	active_fem:				analog_actuator_snapshot;
(*$
	 This message is activated when the active feedback sensor, if present, and  
	analog_actuator <a href="#analog_actuator_status_enum"><i>status</i></a>
 are inchoerent, or it is activated dynamically as a timeout of the activation movement.<br/><br/>
	<a href="#message_behaviour_enum"><i>MESSAGE BEHAVIOUR:</i></a> <i>MESSAGE_BEHAVIOUR_EVENT </i><br/><br/>
	<a href="#machine_reaction_enum"><i>MACHINE REACTION:</i></a> <i>MACHINE_REACTION_NORMAL_STOP </i><br/><br/>
	 The fault codes are specified by ERROR_ID:
	<br/>
	<li> <b>ERRORID_1 = 9</b>: Timeout of activation movement when the <a href="#digital_input_object"><i>di_inactive</i></a>. 
 feedback sensor is covered</li>	
	<li> <b>ERRORID_1 = 10</b>: Timeout of activation movement when the <a href="#digital_input_object"><i>di_ready</i></a>. 
 feedback sensor is not covered</li>	
	<li> <b>ERRORID_1 = 13</b>: Actuator is in <a href="#analog_actuator_status_enum"><i>ANALOG_ACTUATOR_STATUS_ACTIVE</i></a>
 status and the <a href="#digital_input_object"><i>di_ready</i></a> feedback sensor is not covered, or 
 actuator is in <a href="#analog_actuator_status_enum"><i>ANALOG_ACTUATOR_STATUS_INACTIVE</i></a>
 status and the <a href="#digital_input_object"><i>di_ready</i></a> feedback sensor is covered. </li>
$*)

	inactive_fem:			analog_actuator_snapshot;
(*$
	 This message is activated when the inactive feedback sensor, if present, and  
	analog_actuator <a href="#analog_actuator_status_enum"><i>status</i></a>
 are inchoerent, or it is activated dynamically as a timeout of the deactivation movement.<br/><br/>
	<a href="#message_behaviour_enum"><i>MESSAGE BEHAVIOUR:</i></a><i> MESSAGE_BEHAVIOUR_EVENT</i><br/><br/>
	<a href="#machine_reaction_enum"><i>MACHINE REACTION:</i></a><i> MACHINE_REACTION_NORMAL_STOP</i><br/><br/>
	 The fault codes are specified by <i>ERROR_ID</i>:
	<br/>
	<ul>
	<li> <b><i>ERRORID_1 = 11</i></b>: Timeout of deactivation movement when the <a href="#digital_input_object"><i>di_ready</i></a>. 
 feedback sensor is covered</li>	
	<li> <b><i>ERRORID_1 = 12</i></b>: Timeout of deactivation movement when the <a href="#digital_input_object"><i>di_inactive</i></a>. 
 feedback sensor is not covered</li>	
	<li> <b><i>ERRORID_1 = 14</i></b>: Actuator is in <a href="#analog_actuator_status_enum"><i>ANALOG_ACTUATOR_STATUS_INACTIVE</i></a>
 status and the <a href="#digital_input_object"><i>di_inactive</i></a> feedback sensor is not covered, or 
 actuator is in <a href="#analog_actuator_status_enum"><i>ANALOG_ACTUATOR_STATUS_ACTIVE</i></a>
 status and the <a href="#digital_input_object"><i>di_inactive</i></a> feedback sensor is covered. </li>
 </ul>
$*)

	CONVERSION_private:				analog_actuator_private;

    active_elapsed_time: 	LREAL := 0.0;(*$M desc := Elapsed time from the "activate command" and execution finished.; $*)
    deactive_elapsed_time:  LREAL := 0.0;(*$M desc := Elapsed time from the "deactivate command" and execution finished.; $*)

   	ao_setpoint_value: 		LREAL := 0.0;(*$M desc := Analog Output Physical Value; $*)
    ai_feedback_value: 		LREAL := 0.0;(*$M desc := Analog Input Physical Value; $*)

	light_test_active:		BOOL := FALSE;						(*$H_RW desc := Light test is active; $*)

	END_STRUCT
END_TYPE

// ---- Data types/AFL extensions/analog_actuator/analog_actuator_command_enum.TcDUT
TYPE
	analog_actuator_command_enum: (
	ANALOG_ACTUATOR_CMD_NONE			:= 0,	(*$ No command assigned $*)
	ANALOG_ACTUATOR_CMD_INIT			:= 2,	(*$ Initialization command $*)
	ANALOG_ACTUATOR_CMD_ACTIVATE		:= 6,	(*$ Activation command $*)
	ANALOG_ACTUATOR_CMD_DEACTIVATE		:= 8	(*$ Deactivation command $*)
	) := ANALOG_ACTUATOR_CMD_INIT;
END_TYPE

// ---- Data types/AFL extensions/analog_actuator/analog_actuator_fault_reaction_enum.TcDUT
TYPE
	analog_actuator_fault_reaction_enum: (
	ANALOG_ACTUATOR_FAULT_REACTION_DEACTIVATING	:= 0,	(*$ When faulted the analog_actuator sets the
																<a href="#digital_output_object"><i>output</i></a>
																consistently with a deactivate command $*)
	ANALOG_ACTUATOR_FAULT_REACTION_HOLD			:= 1,	(*$ When faulted the analog_actuator sets the
																<a href="#digital_output_object"><i>output</i></a>
																consistently with the current command $*)
	ANALOG_ACTUATOR_FAULT_REACTION_IGNORE		:= 2	(*$ No automatic internal reaction, the application handle the fault condition of analog_actuator $*)
) := ANALOG_ACTUATOR_FAULT_REACTION_DEACTIVATING;
END_TYPE

// ---- Data types/AFL extensions/analog_actuator/analog_actuator_snapshot.TcDUT
(*$S desc := Snapshot; $*)
TYPE
	analog_actuator_snapshot:	STRUCT
	message:        message;

	status:			analog_actuator_status_enum;
	(*$
	Value of the analog_actuator <a href="#analog_actuator_status_enum"><i>status</i></a> field
	when the message is set 
	$*)
	command:		analog_actuator_command_enum;
	(*$
	Value of the analog_actuator <a href="#analog_actuator_command_enum"><i>command</i></a> field
	when the message is set 
	$*)
	is_active:		BOOL;
	(*$
		Value of the active <a href="#digital_input_object"><i>digital_input</i></a>
		when the message is set 
	$*)
	is_inactive:	BOOL;
	(*$
		Value of the inactive <a href="#digital_input_object"><i>digital_input</i></a>
		when the message is set 
	$*)
END_STRUCT
END_TYPE

// ---- Data types/AFL extensions/analog_actuator/analog_actuator_status_enum.TcDUT
(*$ analog_actuator status $*)
TYPE
	analog_actuator_status_enum: (
	ANALOG_ACTUATOR_STATUS_INIT				:= 0,	(*$ analog_actuator initialization $*)
	ANALOG_ACTUATOR_STATUS_ACTIVE 			:= 4,	(*$ analog_actuator is active $*)
	ANALOG_ACTUATOR_STATUS_ACTIVATING		:= 5,	(*$ analog_actuator is executing
														an activation command $*)
	ANALOG_ACTUATOR_STATUS_INACTIVE			:= 6,	(*$ analog_actuator is inactive $*)
	ANALOG_ACTUATOR_STATUS_DEACTIVATING		:= 7,	(*$ analog_actuator is executing
														a deactivation command $*)
	ANALOG_ACTUATOR_STATUS_FAULTED			:= 8	(*$ analog_actuator is in fault status $*)
	) := ANALOG_ACTUATOR_STATUS_INIT;
END_TYPE

// ---- Data types/AFL extensions/analog_actuator/analog_actuator_test.TcDUT
(*$T desc := Test structure; $*)
TYPE
analog_actuator_test:	STRUCT
	command:			analog_actuator_test_command_enum := ANALOG_ACTUATOR_TEST_CMD_IDLE;
															(*$H_W desc := Command (the variable
															  is written by HMI)..; $*)
	command_info:		ARRAY[0..ANALOG_ACTUATOR_MAX_TEST_COMMANDS] OF test_command_info;
															(*$ Structure that informs the HMI
																of the availability of every single
																command and its operational state $*)
    physical_value:		REAL := 0.0;						(*$P min := APPL; max := APPL; step := 0.1;
																 unit := APPL; desc := Analog output physical
																 actual forcing value ; $*)
	
END_STRUCT
END_TYPE

// ---- Data types/AFL extensions/analog_actuator/analog_actuator_test_command_enum.TcDUT
TYPE
	analog_actuator_test_command_enum: (
	ANALOG_ACTUATOR_TEST_CMD_IDLE			:= 0,	(*$ No command assigned $*)
	ANALOG_ACTUATOR_TEST_CMD_ACTIVATE		:= 1,	(*$ Activation command $*)
	ANALOG_ACTUATOR_TEST_CMD_DEACTIVATE		:= 2	(*$ Deactivation command $*)
	) := ANALOG_ACTUATOR_TEST_CMD_IDLE;
END_TYPE

// ---- Data types/AFL extensions/analog_actuator/private/analog_actuator_private.TcDUT
TYPE
	analog_actuator_private :	STRUCT
	initialized:		BOOL := FALSE;		(* The object has been initialized by _init function. *)
	cycle_is_active:	BOOL := FALSE;		(* Cycle function is correctly called. *)
	my_address:			POINTER_TO_VOID; 	(* Object address(pointer).
												Used by HMI for establish
												the objects relations *)

END_STRUCT
END_TYPE

// ---- Data types/AFL extensions/jog_manager/jog_manager.TcDUT
(*   Copyright (c) 2007-2008 G.D SpA
*****************************************************************************************

Date:      Time:     | Author:   				|    Time spent: | Tester:   	   |  Time spent
*****************************************************************************************
*)
(*$
	The <i>jog_manager</i> class abstracts a to manage the axis jog movement.<br/>
	The object is constructed with the <a href="#jog_manager_init"><i>jog_manager_init()</i></a> 
	method and <a href="#axis_object"><i>axi</i></a> are optionally <br/>
	added through the method <a href="#jog_manager_add_axis"><i>jog_manager_add_axis()</i></a>.	
$*)
(* Last used errorID_1 := 15 *)
TYPE
	jog_manager:	STRUCT
	class_name:				STRING(MAX_OBJ_NAME_LENGTH) := JOG_MANAGER_CLASS_NAME;

	object_name:			STRING(MAX_OBJ_NAME_LENGTH) := '';

	descriptor:				descriptor;

	status:					jog_manager_status_enum := JOG_MANAGER_STATUS_INIT;
	(*$M
	desc := Internal status of the jog_manager: value among those defined in the <br/>
	enumerative <a href="#jog_manager_status_enum"><i>jog_manager_status_enum</i></a>; 
	$*)
	command:				jog_manager_command_enum := JOG_MANAGER_CMD_NONE;
												(*$ Command that jog_manager
													is going to execute; value among
													those defined in the enumerative
													jog_manager_command_enum $*)
	operational_command:	jog_manager_command_enum := JOG_MANAGER_CMD_NONE;
												(*$ Command assigned when jog_manager
													is in the "operational" mode; value among
													those defined in the enumerative
													jog_manager_command_enum $*)
	test:					jog_manager_test;
												(*$ This struct contains all the test's informations $*)
	parents:				ARRAY[1..JOG_MANAGER_MAX_PARENTS] OF POINTER TO jog_manager;												
	parents_next_free:		UINT;
												(*$ This array contains all the parent jog_manager $*)
	axis_list:				ARRAY[JOG_MANAGER_JOG_LIST_NONE..JOG_MANAGER_JOG_LIST_MAX] OF jog_manager_element;
												(*$ This struct contains all the axis_jog information $*)
	jog_activation_condition: BOOL;
												(*$ Jog activation condition $*)			
	jog_active:				BOOL;				
	(*$P desc := jog mode active; $*)
	jog_active_pow:			parameter_overwrite;
	(*$I desc := Parameter overwite to inizialithe the value at startup; $*)
	enable_sw_limit:		BOOL;				
	(*$P desc := software limit active; $*)	
	enable_sw_limit_pow:	parameter_overwrite;
	(*$I desc := Parameter overwite to adjust the SW limit check; $*)																										
	axis_act_position_linear: LREAL;
	(*$M unit := mm;
		desc := currently selected axis position; 
	$*)
	axis_act_position_rotative: LREAL;
	(*$M unit := °;
		desc := currently selected axis position; 
	$*)		
	axis_act_torque_rotative: LREAL;
	(*$M unit := %;
		desc := currently selected axis torque (the value is axis indipendent! it's doubled for management reason!; 
	$*)
	axis_act_torque_linear: LREAL;
	(*$M unit := %;
		desc := currently selected axis torque (the value is axis indipendent! it's doubled for management reason!; 
	$*)	
	axis_cmd_position_linear: LREAL;
	(*$P min :=  -1000; max :=  2000; step := 1; unit := mm/s;
		desc := jog command position (linear jog axis); 
	$*)
	axis_cmd_position_rotative:	LREAL;
	(*$P min :=  -360; max :=  360; step := 1; unit := °/s;
		desc := jog command position (rotative jog axis); 
	$*)
	axis_cmd_position_rotative_pow:	parameter_overwrite;
	(*$I desc := Parameter overwite to adjust jog command position (rotative); $*)	
	axis_speed_linear:		LREAL;
	(*$P min :=  0; max :=  100; step := 1; unit := mm/s;
		desc := jog speed (linear jog axis); 
	$*)
	axis_cmd_position_linear_pow: parameter_overwrite;
	(*$I desc := Parameter overwite to adjust jog command position (linear); $*)		
	axis_speed_rotative:	LREAL;
	(*$P min :=  0; max :=  100; step := 1; unit := °/s;
		desc := jog speed (rotative jog axis); 
	$*)	
	di_pendant_positive:	POINTER TO digital_input;
	(*$U
	desc := Reference to the <a href="#digital_input_object"><i>digital_input</i></a>
	which refere to jog positive pendant command; 
	$*)
	di_pendant_negative:	POINTER TO digital_input;
	(*$U
	desc := Reference to the <a href="#digital_input_object"><i>digital_input</i></a>
	which refere to jog negative pendant command; 
	$*)
	has_pendant:			BOOL;
												(*$ Pendant present $*)
	pendant_active:			BOOL;				
	(*$P desc := pendant active; $*)
	pendant_active_pow:		parameter_overwrite;
	(*$I desc := Parameter overwite to inizialithe the value at startup; $*)
	has_shared_pendant:		POINTER TO jog_manager;
	(*$ Pointer to jog_manager instance that manage directly the pendant $*)
	shared_pendant_active:	BOOL;	
	(*$ Shared pendant activation status $*)
								
	hmi_jog_positive_cbtn:	command_button;		(*$I expose{ value_from_hmi; button_status.status; button_led.color; button_led.graphic_object.status;} desc := jog plus; $*)
	hmi_jog_negative_cbtn:	command_button;		(*$I expose{ value_from_hmi; button_status.status; button_led.color; button_led.graphic_object.status;} desc := jog minus; $*)
	hmi_jog_absolute_cbtn:	command_button;		(*$I expose{ value_from_hmi; button_status.status; button_led.color; button_led.graphic_object.status;} desc := jog absolute; $*)
	hmi_jog_selection_hgos:	hmi_graphic_object_status;	(*$I expose{ status;} desc := enable jog selection; $*)
	hmi_rot_selection_hgos: hmi_graphic_object_status;	(*$I expose{ status;} desc := enable linear axis; $*)
	hmi_lin_selection_hgos: hmi_graphic_object_status;	(*$I expose{ status;} desc := enable rotative axis; $*)
	hmi_sw_limit_hgos: 		hmi_graphic_object_status;	(*$I expose{ status;} desc := enable sw limit; $*)
	hmi_pendant_active_hgos:hmi_graphic_object_status;	(*$I expose{ status;} desc := enable pendant selection; $*)
	hmi_pendant_positive_ld:led;						(*$I expose{ color; graphic_object.status;} desc := pendant positive status; $*)
	hmi_pendant_negative_ld:led;						(*$I expose{ color; graphic_object.status;} desc := pendant negative status; $*)
	
	CONVERSION_private:		jog_manager_private;
												(*$ Private struct $*)
	END_STRUCT
END_TYPE

// ---- Data types/AFL extensions/jog_manager/jog_manager_command_enum.TcDUT
TYPE
	jog_manager_command_enum: (
	JOG_MANAGER_CMD_NONE						:= 0,	(*$ No command assigned $*)
	JOG_MANAGER_SET_ACTIVATION_CONDITION		:= 1,
	JOG_MANAGER_RESET_ACTIVATION_CONDITION		:= 2,
	JOG_MANAGER_STOP_ABSOLUTE_MOVEMENT			:= 3
	) := JOG_MANAGER_CMD_NONE;
END_TYPE

// ---- Data types/AFL extensions/jog_manager/jog_manager_element.TcDUT
TYPE jog_manager_element : 
STRUCT
	axis:					POINTER TO axis;
	master_axis:			BOOL := FALSE;	
	jog_type:				jog_manager_type := JOG_TYPE_NONE;	
	sw_limit_positive:		LREAL := 0.0; //No check if both zero!
	sw_limit_negative:		LREAL := 0.0;
	all_slave_axis_engaged:	BOOL := FALSE;	
END_STRUCT
END_TYPE

// ---- Data types/AFL extensions/jog_manager/jog_manager_snapshot.TcDUT
(*$S desc := Snapshot; $*)
TYPE
	jog_manager_snapshot:	STRUCT
	message:        message;

	status:			jog_manager_status_enum;
	(*$
	Value of the jog_manager <a href="#jog_manager_status_enum"><i>status</i></a> field
	when the message is set 
	$*)
	command:		jog_manager_command_enum;
	(*$
	Value of the jog_manager <a href="#jog_manager_command_enum"><i>command</i></a> field
	when the message is set 
	$*)	
END_STRUCT
END_TYPE

// ---- Data types/AFL extensions/jog_manager/jog_manager_status_enum.TcDUT
(*$ jog_manager status $*)
TYPE
	jog_manager_status_enum: (
	JOG_MANAGER_STATUS_INIT						:= 0,	(*$ jog_manager initialization $*)
	JOG_MANAGER_STATUS_IDLE						:= 1,	(*$ jog_manager idle status $*)
	JOG_MANAGER_STATUS_READY					:= 2,	(*$ jog_manager ready to select jog mode $*)
	JOG_MANAGER_STATUS_ACTIVE					:= 3,	(*$ jog_manager jog mode active $*)
	JOG_MANAGER_STATUS_SEL_DISABLE_AXIS			:= 10,	(*$ jog_manager disable selected axis $*)
	JOG_MANAGER_STATUS_OLD_DISABLE_AXIS			:= 11,	(*$ jog_manager disable previous axis $*)
	JOG_MANAGER_STATUS_SEL_ENABLE_AXIS			:= 20,	(*$ jog_manager enable selected axis $*)
	JOG_MANAGER_STATUS_SEL_ENABLED_AXIS			:= 21,	(*$ jog_manager enabled selected axis $*)
	JOG_MANAGER_STATUS_LINEAR_JOG_POSITIVE		:= 31,	(*$ jog_manager jog+ linear $*)
	JOG_MANAGER_STATUS_LINEAR_JOG_NEGATIVE		:= 32,	(*$ jog_manager jog- linear $*)
	JOG_MANAGER_STATUS_ROTATIVE_JOG_POSITIVE	:= 33,	(*$ jog_manager jog+ rotative $*)
	JOG_MANAGER_STATUS_ROTATIVE_JOG_NEGATIVE	:= 34,	(*$ jog_manager jog+ rotative $*)
	JOG_MANAGER_STATUS_ABSOLUTE_STARTING		:= 40,	(*$ jog_manager jog absolute starting $*)
	JOG_MANAGER_STATUS_ABSOLUTE_MOVING			:= 41,	(*$ jog_manager jog absolute moving $*)
	JOG_MANAGER_STATUS_STOP_ABSOLUTE_MOVING		:= 42,	(*$ jog_manager stop absolute moving $*)
	JOG_MANAGER_STATUS_STOPPING					:= 50	(*$ jog_manager stopping $*)
	) := JOG_MANAGER_STATUS_INIT;
END_TYPE

// ---- Data types/AFL extensions/jog_manager/jog_manager_test.TcDUT
(*$T desc := Test structure; $*)
TYPE
jog_manager_test:	STRUCT
	command:			jog_manager_test_command_enum := JOG_MANAGER_TEST_CMD_NONE;
															(*$H_W desc := Command (the variable
															  is written by HMI)..; $*)
	command_info:		ARRAY[0..JOG_MANAGER_MAX_TEST_COMMANDS] OF test_command_info;
															(*$ Structure that informs the HMI
																of the availability of every single
																command and its operational state $*)    
END_STRUCT
END_TYPE

// ---- Data types/AFL extensions/jog_manager/jog_manager_test_command_enum.TcDUT
TYPE
	jog_manager_test_command_enum: (
	JOG_MANAGER_TEST_CMD_NONE				:= 0	(*$ No command assigned $*)
	) := JOG_MANAGER_TEST_CMD_NONE;
END_TYPE

// ---- Data types/AFL extensions/jog_manager/jog_manager_type.TcDUT
TYPE jog_manager_type :
(
	JOG_TYPE_NONE 				:= 0,
	JOG_TYPE_ROTATIVE			:= 1,
	JOG_TYPE_ROTATIVE_PLUS		:= 2,
	JOG_TYPE_ROTATIVE_MINUS		:= 3,
	JOG_TYPE_LINEAR				:= 10,
	JOG_TYPE_LINEAR_PLUS		:= 11,
	JOG_TYPE_LINEAR_MINUS		:= 12
) := JOG_TYPE_NONE;
END_TYPE

// ---- Data types/AFL extensions/jog_manager/private/jog_manager_private.TcDUT
TYPE
	jog_manager_private :	STRUCT
	initialized:		BOOL := FALSE;		(* The object has been initialized by _init function. *)
	cycle_is_active:	BOOL := FALSE;		(* Cycle function is correctly called. *)
	my_address:			POINTER_TO_VOID; 	(* Object address(pointer).
												Used by HMI for establish
												the objects relations *)
																	
	jog_pendant_positive:				BOOL;
	jog_pendant_negative:				BOOL;
		
	axis_is_absolute_moving:			BOOL;
	axis_absolute_moving_direction:		axis_direction_enum;
			
	update_parameters:					UINT;							
	list_selected:						UINT;												
	list_selected_is_valid:				BOOL;
	list_selected_axis_is_valid:		BOOL;													
	old_list_selected:					UINT;
	old_list_selected_is_valid:			BOOL;
	old_list_selected_axis_is_valid:	BOOL;							
	sw_limit_active:					BOOL;
	sw_limit_active_positive:			BOOL;
	sw_limit_active_negative:			BOOL;
	axis_is_linear:						BOOL;
	axis_is_rotative:					BOOL;
	jog_positive_enable:				BOOL;
	jog_negative_enable:				BOOL;
	
	shared_pendant_jog_positive_status:	BOOL;
	shared_pendant_jog_negative_status:	BOOL;
END_STRUCT
END_TYPE

// ---- Data types/Common/plc_target_type_enum.TcDUT
TYPE plc_target_type_enum :
(
	PLC_TARGET_MACHINE 			:= 0, 		(*PLC works connected to a real machine*)
	PLC_TARGET_LOCAL 			:= 1,		(*PLC works connected to a local simulator*)
	PLC_TARGET_LOCAL_IP			:= 2		(*PLC works connected to a local simulator with Industrial Physics*)
) := PLC_TARGET_LOCAL;

END_TYPE

// ---- POUs/AFL extensions/IO_Link/bis00lh/iol_slave_bis00lh_bitheader_input.TcDUT
TYPE iol_slave_bis00lh_bitheader_input :
STRUCT
	CP: BIT;
	AA: BIT;
	AE: BIT;
	AF: BIT;
	///unused
	Bit4: BIT;
	_TO: BIT;
	HF: BIT;
	BB: BIT;
END_STRUCT
END_TYPE

// ---- POUs/AFL extensions/IO_Link/bis00lh/iol_slave_bis00lh_bitheader_output.TcDUT
TYPE iol_slave_bis00lh_bitheader_output :
STRUCT
	AV: BIT;
	///unused
	Bit1: BIT;
	GR: BIT;
	///unused
	Bit3: BIT;
	///unused
	Bit4: BIT;
	KA: BIT;
	TI: BIT;
	///unused
	Bit7: BIT;
END_STRUCT
END_TYPE

// ---- POUs/AFL extensions/IO_Link/bis00lh/iol_slave_bis00lh_data.TcDUT
TYPE iol_slave_bis00lh_data :
STRUCT
	a:bool; (*To remove LB issue*)
END_STRUCT
END_TYPE

// ---- POUs/AFL extensions/IO_Link/bis00lh/iol_slave_bis00lh_pdo_input.TcDUT
TYPE	iol_slave_bis00lh_pdo_input :		
STRUCT
	DeviceDiag AT %I*: BOOL;
	DeviceState AT %I*: BOOL;
	ChannelState AT %I*: USINT;
	InfoDataState AT %I*: UINT;
	ByteArr AT %I*: ARRAY[0..9] OF BYTE;
END_STRUCT
END_TYPE

// ---- POUs/AFL extensions/IO_Link/bis00lh/iol_slave_bis00lh_pdo_output.TcDUT
TYPE	iol_slave_bis00lh_pdo_output :		
STRUCT
		ByteArr AT %Q*: ARRAY[0..9] OF BYTE;
END_STRUCT
END_TYPE

// ---- POUs/AFL extensions/IO_Link/ml2prime/iol_slave_mlg2prime_output_status_1.TcDUT
TYPE iol_slave_mlg2prime_output_status_1 :
STRUCT
	q1:							BIT;
	q2:							BIT;
	q3:							BIT;
	q4:							BIT;	
END_STRUCT
END_TYPE

// ---- POUs/AFL extensions/IO_Link/ml2prime/iol_slave_mlg2prime_system_status_1.TcDUT
TYPE iol_slave_mlg2prime_system_status_1 :
STRUCT
	sync_error:					BIT;
	teach_fail:					BIT;
	hardware_error:				BIT;
	contamination_alarm:		BIT;
	teach_active:				BIT;
	over_temp:					BIT;
	data_invalid:				BIT;
	q_short_circuit:			BIT;
END_STRUCT
END_TYPE

// ---- POUs/AFL extensions/IO_Link/Struct/iol_slave_bsp00ue_data.TcDUT

TYPE
	iol_slave_bsp00ue_data :		STRUCT
	setpoint:						DWORD; 
	switchpoint:					DWORD; 
	measure_unit:					BYTE; 
	max_press:						WORD; 
	min_press:						WORD; 
	switchpoint_delay_on:			WORD; 
	switchpoint_delay_off:			WORD; 
	measure_damping:				WORD; 
END_STRUCT
END_TYPE

// ---- POUs/AFL extensions/IO_Link/Struct/iol_slave_mlg2prime_data.TcDUT

TYPE
	iol_slave_mlg2prime_data:				STRUCT

	teach_in_state:                   		SINT;		
	quality_of_teach:						BYTE;
	quality_of_run:							BYTE;
	teach_result:							BYTE;
	StdQA1Configuration:         			INT;		
	CrossBeamEnable:						BYTE;		
	temperature:							BYTE;		
	system_status:							BYTE;
	device_status:							BYTE;
	blanking_teach_enable:					BYTE;
END_STRUCT
END_TYPE

// ---- POUs/AFL extensions/IO_Link/Struct/iol_slave_ray26p_data.TcDUT

TYPE
	iol_slave_ray26p_data:					STRUCT

	teach_in_state:                   		BYTE;		
	set_inverted_logic:						BYTE;		
	actual_inverted_logic:					BYTE;		
	quality_of_teach:						BYTE;
	teach_in_channel:						BYTE;
	system_state:							BYTE;
	sender_configuration:					BYTE;
	Pin2_configuration:						BYTE;
END_STRUCT
END_TYPE

// ---- Global Variables/AFL extensions/analog_actuator_global.TcGVL
{attribute 'Tc2GvlVarNames'}
VAR_GLOBAL CONSTANT
	(* analog_actuator define *)
	ANALOG_ACTUATOR_CLASS_NAME:		STRING := 'analog_actuator';
	ANALOG_ACTUATOR_MAX_TEST_COMMANDS:	DINT :=	2;
END_VAR

VAR_GLOBAL
END_VAR

// ---- Global Variables/AFL extensions/jog_manager_global.TcGVL
{attribute 'Tc2GvlVarNames'}
VAR_GLOBAL CONSTANT
	(* jog_manager define *)
	JOG_MANAGER_CLASS_NAME:			STRING := 'jog_manager';
	JOG_MANAGER_MAX_TEST_COMMANDS:	DINT :=	0;
	JOG_MANAGER_MAX_PARENTS:		UINT := 10;
	
	JOG_MANAGER_JOG_LIST_NONE:		UINT := 0;
	JOG_MANAGER_JOG_LIST_MAX:		UINT := 100;
	
	SW_LIMIT_LINEAR_POSITIVE:		LREAL := 2000.0;
	SW_LIMIT_LINEAR_NEGATIVE:		LREAL := -1000.0;
	SW_LIMIT_ROTATIVE_POSITIVE:		LREAL := 180.0;
	SW_LIMIT_ROTATIVE_NEGATIVE:		LREAL := -180.0;
END_VAR

VAR_GLOBAL
END_VAR

// ---- Global Variables/Application/Common/common_global_variables.TcGVL
(*********************************** G.D S.p.A. - Technical Department ***********************************
============= PROGRAM INFO ============


============= DESCRIPTION =============
Application common global variables list

============= REVISIONS ===============
Date		Version	 	Author      	Description             
----------	-------		------------  	--------------------------------------------
2019/04/18 	0000.00	 	G.Cera 			Creation of the PRG
**********************************************************************************************************)
{attribute 'Tc2GvlVarNames'}
VAR_GLOBAL CONSTANT

(*	ITEM_ABSENT:										DWORD := 16#0000_0000;
	ITEM_TO_REJECT:										DWORD := 16#0000_0001;
	ITEM_REJECTED:										DWORD := 16#0000_0002;
	ITEM_PRESENT:										DWORD := 16#0000_0003;
*)
    NONE:												DWORD := 16#0000_0000;
    ALL:												DWORD := 16#FFFF_FFFF;
    DWORD_BIT_0	:										DWORD := 16#0000_0001;
	
	ITEM_CASE_FEED:										DWORD := ITEM_AUX_BIT_4;
	ITEM_HAS_CARTON:									DWORD := ITEM_AUX_BIT_5;
	ITEM_HAS_LS_UPPER_FLAP:								DWORD := ITEM_AUX_BIT_6;
	ITEM_HAS_LS_LOWER_FLAP:								DWORD := ITEM_AUX_BIT_7;
	ITEM_HAS_OS_UPPER_FLAP:								DWORD := ITEM_AUX_BIT_8;
	ITEM_HAS_OS_LOWER_FLAP:								DWORD := ITEM_AUX_BIT_9;
	(*ITEM_HAS_GLUE_ON_CASE:								DWORD := ITEM_AUX_BIT_9;*)
	ITEM_HAS_LS_UPPER_FLAP_AT_GLUE:						DWORD := ITEM_AUX_BIT_10;
	ITEM_HAS_OS_UPPER_FLAP_AT_GLUE:						DWORD := ITEM_AUX_BIT_11;
	ITEM_HAS_OPEN_FLAP_LS:								DWORD := ITEM_AUX_BIT_12;
	ITEM_HAS_OPEN_FLAP_OS:								DWORD := ITEM_AUX_BIT_13;
	ITEM_POWER_UP:										DWORD := ITEM_AUX_BIT_14;
	ITEM_HAS_LOAD:										DWORD := ITEM_AUX_BIT_15;
	ITEM_HAS_TRANSFER_LOAD_BUILD_COMPLETE:				DWORD := ITEM_AUX_BIT_16;
	
	(* SHIFT REGISTER IDENTITY CARD *)
	(*****************************)
	
	(* MOTION *)
	G_VIRTUAL_ENCODER_SCALING_FACTOR_DEGPINC:			LREAL := 1.0;
	G_SERVO_ENCODER_SCALING_FACTOR_DEGPINC:				LREAL := 0.0001;	
	G_NO_MODULO_DEG:									LREAL := 0;
	G_MODULO_360_DEG:									LREAL := 360;	
	G_MODULO_720_DEG:									LREAL := 720;
	G_MODULO_1080_DEG:									LREAL := 1080;
	G_MODULO_4320_DEG:									LREAL := 4320;

	G_CONV_S_TO_MS:										INT := 1000;
	G_CONV_PPM_TO_DEGPS:								LREAL := 6.0;
	G_CONV_KG_TO_NM:									LREAL := 9.80665;	

	MAX_INT_VALUE:										INT := 32767;		(* Global_Variables: 32767*)
	MIN_INT_VALUE:										INT := -32768;		(* Global_Variables: -32768*)
	MAX_WORD_VALUE:										WORD := 65535;		(* Global_Variables: 65535*)

	WORD_MASK_HIGH_BYTE:								WORD := 16#FF00;	(* Global_Variables: Maschera x WORD elimina la parte bassa *)
	WORD_MASK_LOW_BYTE:									WORD := 16#00FF;	(* Global_Variables: Maschera x WORD elimina la parte alta *)

	CUPS_NUMBER_PICKED_BY_R1_R2:						INT := 12;
	CUPS_FEEDING_CROSS_SECTION_ENABLE_PHASE:			INT := 190;
	PICK_AND_PLACE_ROBOTS_NUMBER:						INT := 6;
END_VAR


VAR_GLOBAL
	(* MACHINE CONFIGURATION *)
	//sw_configurator:									sw_configurator_struct;		
	csp_sw_configurator:									csp_sw_configurator_struct;	

	(* APPLICATION STATUS *)
	g_application_status_1st_powerup_high:				BOOL;
	g_application_status_1st_powerup_normal:			BOOL;
	g_application_status_1st_powerup_low:				BOOL;

	g_application_status_2nd_powerup_high:				BOOL;
	g_application_status_2nd_powerup_normal:			BOOL;
	g_application_status_2nd_powerup_low:				BOOL;

	g_application_status_3rd_powerup_high:				BOOL;
	g_application_status_3rd_powerup_normal:			BOOL;
	g_application_status_3rd_powerup_low:				BOOL;

	g_application_status:								application_status_enum;
	
	power_done:											BOOL := FALSE;
	(*PLC_TARGET_MACHINE, PLC_TARGET_LOCAL, PLC_TARGET_LOCAL_IP *)
	g_plc_target:										plc_target_type_enum := PLC_TARGET_LOCAL;
	
	RAJ_to_Flexlink AT %Q*:							ARRAY[0..3] OF DINT;
	Flexlink_to_RAJ AT %I*:							ARRAY[0..3] OF DINT;
	RAJ_to_Cartoner AT %Q*:							ARRAY[0..19] OF DINT;
	Cartoner_to_RAJ AT %I*: 						ARRAY[0..19] OF DINT;
	
END_VAR

VAR_GLOBAL RETAIN
	g_application_status_1st_powerup_high_absolute:		BOOL:=FALSE;
	g_application_status_1st_powerup_normal_absolute:	BOOL:=FALSE;
	g_application_status_1st_powerup_low_absolute:		BOOL:=FALSE;
END_VAR

VAR_GLOBAL PERSISTENT
	csp_retain_data:									csp_retain_data_struct;
END_VAR

// ---- Application/_Tasks/_highest.TcPOU
(*********************************** G.D S.p.A. - Technical Department ***********************************
============= PROGRAM INFO ============
FOLDER:             TBD
MACHINES INVOLVED:  TBD 

============= DESCRIPTION =============
Highest task

============= REVISIONS ===============
Date		Version	 	Author      	Description             
----------	-------		------------  	--------------------------------------------
2019/04/05 	0000.00	 	G.Cera 			Creation of the PRG

**********************************************************************************************************)
{attribute 'TcCallAfterOutputUpdate'}
PROGRAM _highest
VAR
END_VAR

(* APPLICATION *)
framework_highesttask_begin();

//application_status_manager();
application_status_manager_highest();

_csp_highest();

//dbg_highest();

framework_highesttask_end();

END_PROGRAM

// ---- Application/_Tasks/Application Status Manager/application_status_manager_highest.TcPOU
(********************* G.D S.p.A. - Technical Department ***********************************
Date        Version Author      	Description             
----------  ------- ----------- 	--------------------------------------------------------
2019/04/23	0000.01	G.Cera			Creation of the POU

DESCRIPTION:
Manager of the application status high. it is called by highest speed task


NOTES:

********************************************************************************************)
PROGRAM application_status_manager_highest
VAR

END_VAR

VAR_OUTPUT

END_VAR

IF g_application_status=APPLICATION_STATUS_1ST_POWERUP_ABSOLUTE
THEN
   	g_application_status_1st_powerup_high_absolute:=TRUE;
END_IF

IF g_application_status=APPLICATION_STATUS_1ST_POWERUP
THEN
   	g_application_status_1st_powerup_high:=TRUE;
END_IF

IF g_application_status=APPLICATION_STATUS_2ND_POWERUP
THEN
   	g_application_status_2nd_powerup_high:=TRUE;
END_IF

IF g_application_status=APPLICATION_STATUS_3RD_POWERUP
THEN
   	g_application_status_3rd_powerup_high:=TRUE;
END_IF;

END_PROGRAM

// ---- Application/CSP/_Tasks/_csp_highest.TcPOU
(*********************************** G.D S.p.A. - Technical Department ***********************************
============= PROGRAM INFO ============
FOLDER:             TBD
MACHINES INVOLVED:  TBD 

============= DESCRIPTION =============
CSP: highest task

============= REVISIONS ===============
Date		Version	 	Author      	Description             
----------	-------		------------  	--------------------------------------------
2019/04/05 	0000.00	 	G.Cera 			Creation of the PRG

**********************************************************************************************************)

PROGRAM _csp_highest
VAR
END_VAR


IF g_application_status = APPLICATION_STATUS_RUNNING
THEN
	IF message_is_on(csp.mch.cpu_startup_aem.message)
	THEN
			power_done := TRUE;
	END_IF
END_IF

_csp_case_highest();

_csp_transfer_highest();

_csp_main_highest();

_csp_customerInterfaces_highest();

END_PROGRAM

// ---- Application/CSP/csp.TcPOU
(*********************************** G.D S.p.A. - Technical Department ***********************************
============= PROGRAM INFO ============
FOLDER:             TBD
MACHINES INVOLVED:  TBD 

============= DESCRIPTION =============
csp machine declaration

============= REVISIONS ===============
Date		Version	 	Author      	Description             
----------	-------		------------  	--------------------------------------------
2019/04/05 	0000.00	 	M.Grasso		Creation of the PRG

**********************************************************************************************************)

PROGRAM csp
VAR
	mch:						machine;
	reset_timer:				timer;
	start_timer:				timer;
	
		
	restart_bit: 				BOOL;
	TC_Restart1:				TC_Restart;
	DriveCommFailureTON: 		TON;
	DriveCommFailure:			BOOL := FALSE;
	DriveCommFailurePT: 		TIME := T#1M;
	DriveCommFailed_RestartPC: 	BOOL := FALSE;
	FB_EcSetMasterState1:		FB_EcSetMasterState;

END_VAR

VAR_INPUT
	i_reset_button:			BOOL;
	i_start_button:			BOOL;
END_VAR

VAR_OUTPUT
	o_machine_is_ready:		BOOL;
	o_machine_is_running:	BOOL;
	o_machine_is_stopped:	BOOL;
	o_machine_is_emergency_stopped:	BOOL;
END_VAR

_read_var_input();

_object_manager();

IF NOT objects_running()
THEN
	RETURN;	
END_IF

_read_process_image();

_mode_manager();

_set_runtime_properties();

(********************************* BODY *********************************)
(* MACHINE COMMANDS *)

IF 	(i_reset_button
	OR
	csp_case_main_services_pushbuttons.reset_pressed
	OR
	csp_transfer_main_services_pushbuttons.reset_pressed) // 8/28
	AND
	machine_is_stopped(mch)
	AND
	csp_main_services_pushbuttons.reset_delay_ton_complete1 //timer_is_expired(csp_main_services_pushbuttons.reset_tmr)
THEN
	machine_reset(mch);
	
END_IF

IF 	i_start_button
	AND
	csp_main_services_pushbuttons.start_ton.Q
	AND
	machine_is_ready(mch)
THEN
	machine_start(mch);
END_IF

IF 	hmi_is_connected(mch)
	AND 
	(
		(* If any of the drives/motors are in a faulted Ethercat State with 460V on, restart Twincat to re-establish comms
			Fix for an operator powering off 460V and back on without cycling 24V after. Correct power cycle is 460V then 24V disconnect *)
		(	
			(* Check to see if IO Data Invalid *)
			csp_case_feed_arm_elbow.axis.ax_ref.Status.IoDataInvalid
			AND
			(* Check to see if the drive status has an Ethercat Fault *)
			csp_case_main_drives.SD8200_drv.status = SOE_DRIVE_STATUS_NET_FAULT
			AND
			(* Link_state_is_ok is TRUE when 460V is present *)
			csp_case_main_drives.SD8200_drv.net_ethercat_slave^.link_state_is_ok
		)
		OR
		(	
			(* Check to see if IO Data Invalid *)
			csp_case_transport_os_leading.axis.ax_ref.Status.IoDataInvalid
			AND
			(* Check to see if the drive status has an Ethercat Fault *)
			csp_case_main_drives.SD2100_drv.status = SOE_DRIVE_STATUS_NET_FAULT
			AND
			(* Link_state_is_ok is TRUE when 460V is present *)
			csp_case_main_drives.SD2100_drv.net_ethercat_slave^.link_state_is_ok
		)
		OR
		(	
			(* Check to see if IO Data Invalid *)
			csp_case_fc_ls_upper_follower.axis.ax_ref.Status.IoDataInvalid
			AND
			(* Check to see if the drive status has an Ethercat Fault *)
			csp_case_main_drives.SD10300_drv.status = SOE_DRIVE_STATUS_NET_FAULT
			AND
			(* Link_state_is_ok is TRUE when 460V is present *)
			csp_case_main_drives.SD10300_drv.net_ethercat_slave^.link_state_is_ok
		)
	)
THEN
	DriveCommFailure := TRUE;
ELSE
	DriveCommFailure := FALSE;
END_IF

DriveCommFailureTON(IN:= DriveCommFailure , PT:=DriveCommFailurePT , Q=> DriveCommFailed_RestartPC , ET=> );		

TC_Restart1(
	NETID := '',
	RESTART := DriveCommFailed_RestartPC,
	TMOUT := T#10S);
(************************************************************************)

_handle_messages();

_write_output();

ACTION _handle_messages:
;
END_ACTION

ACTION _handle_process_test:
;
END_ACTION

ACTION _mode_manager:
;
END_ACTION

ACTION _object_manager:
IF 	NOT objects_running()
THEN
	csp_interface_configuration(
		motman					:= csp_main_motorization_manager.motm,
		machine					:= csp.mch,
		CONVERSION_this			:= csp_sw_configurator.csp_INTERFACE);
END_IF

IF 	objects_initialization()
THEN
	machine_init(
		object_name				:= 'csp.mch', 
		name_to_hmi				:= 'Case Packer', 
		CONVERSION_this			:= mch);
END_IF
END_ACTION

ACTION _read_process_image:
;
END_ACTION

ACTION _read_var_input:
i_reset_button	:= csp_main.o_reset_button;
i_start_button	:= csp_main.o_start_button;;
END_ACTION

ACTION _set_runtime_properties:
;
END_ACTION

ACTION _write_output:
o_machine_is_running	:= machine_is_execute(mch) OR motorization_manager_is_held(csp_main_motorization_manager.motm);
o_machine_is_ready		:= machine_is_ready(mch);
o_machine_is_stopped	:= machine_is_stopped(csp.mch);
o_machine_is_emergency_stopped	:= machine_is_stop_emergency_active(csp.mch);
END_ACTION

END_PROGRAM

// ---- Application/CSP/Main/Services/Pushbuttons/csp_main_services_pushbuttons.TcPOU
(*********************************** G.D S.p.A. - Technical Department ***********************************
============= PROGRAM INFO ============
FOLDER:             TBD
MACHINES INVOLVED:  TBD 

============= DESCRIPTION =============
csp main keyboard

============= REVISIONS ===============
Date		Version	 	Author      	Description             
----------	-------		------------  	--------------------------------------------
2019/04/05 	0000.00	 	M.Grasso		Creation of the PRG

**********************************************************************************************************)
(*$R
	process_ref := prc;
$*)
PROGRAM csp_main_services_pushbuttons
VAR
	prc:									process;
	prc_path:				STRING;
	
	reset_request_rtrig:							R_TRIG;
	reset_request:									BOOL;
	reset_tmr:										timer;
	reset_delay:									UDINT;
	
	start_request_rtrig:							R_TRIG;
	start_request:									BOOL;
	start_tmr:										timer;
	start_delay:									UDINT := 5000;
	start_ton:										TON;
	
	immediate_stop_bool:							boolean;
	stop_button_rtrig:								R_TRIG;

	wait_immediate_stop_dvr:						BOOL;
	immediate_stop_dchk: 							digital_check;
	
	stop_dchk_transfer_dvr: 						BOOL;
	stop_dchk_case_dvr: 							BOOL;	
	stopped_bool:									BOOL;
	
	reset_delay_bool: 								BOOL;
	reset_delay_ton1:								TON;
	reset_delay_ton_complete1:						BOOL;
	
	stop_message_reclassification_instance:			message_reclassification;
	unlock_guard_enable_from_reclassification:		BOOL;
	powerup:										BOOL := TRUE;
	service_stop_force_unlock_flt:					filter;

END_VAR

VAR_INPUT
	i_reset_button:			BOOL;
	i_start_button:			BOOL;
	i_stop_button:			BOOL;
	(*PART TO BE MOVED TO MAIN*)
	reset_lamp_on:				BOOL;
	reset_lamp_blink:			BOOL;
	start_lamp_on:				BOOL;
	start_lamp_blink:			BOOL;
	stop_lamp_on:				BOOL;
	stop_lamp_blink:			BOOL;
	(*END PART TO BE MOVED TO MAIN*)
END_VAR

VAR_OUTPUT
	o_machine_is_running:	BOOL;
END_VAR

_read_var_input();

_object_manager();

IF NOT objects_running()
THEN
	RETURN;	
END_IF

_read_process_image();

_mode_manager();

CASE process_get_mode(prc) OF
	MODE_ABSENT,
	MODE_INACTIVE:
		RETURN;
	MODE_TEST:
		_handle_process_test();
END_CASE

_set_runtime_properties();

(********************************* BODY *********************************)
(*Light Logic*)

(*STOP LOGIC *)

boolean_reset(immediate_stop_bool);

IF  (
        NOT stop_dchk_case_dvr
		OR
		NOT stop_dchk_transfer_dvr
    )
    AND
    (
        motorization_manager_is_stopping(csp_main_motorization_manager.motm)
        OR
        motorization_manager_is_emptying(csp_main_motorization_manager.motm)
    )
THEN
    digital_check_enable(immediate_stop_dchk);
    IF  (
            stop_button_rtrig.Q
            AND
            wait_immediate_stop_dvr
        )
    THEN
        boolean_set(immediate_stop_bool);
    END_IF;
    wait_immediate_stop_dvr := TRUE;
END_IF


IF  motorization_manager_is_stopped(CONVERSION_this:= csp_main_motorization_manager.motm)
THEN
    digital_check_disable(immediate_stop_dchk);
    wait_immediate_stop_dvr := FALSE;
END_IF


(* RESET LOGIC *)
IF machine_is_stopped(csp.mch)
AND reset_delay_ton_complete1//timer_is_expired(reset_tmr) // ADDED TO DELAY RESET
THEN
	IF
		motorization_manager_is_stopping(csp_main_motorization_manager.motm)
		OR
		motorization_manager_is_emptying(csp_main_motorization_manager.motm)
	THEN
		reset_lamp_blink := TRUE;
		reset_lamp_on := FALSE;
	ELSE
		reset_lamp_blink := FALSE;
		reset_lamp_on := TRUE;	
	END_IF
ELSE
	reset_lamp_blink := FALSE;
	reset_lamp_on := FALSE;			
END_IF


(* START LOGIC *)
start_ton(
	IN := machine_is_ready(csp.mch),
	PT := UDINT_TO_TIME(start_delay));

(*IF	machine_is_ready(csp.mch)
AND timer_is_expired(start_tmr)*) // ADDED TO DELAY START
IF start_ton.Q
THEN
	start_lamp_blink := FALSE;
	start_lamp_on := TRUE;
ELSIF motorization_manager_is_suspended(csp_main_motorization_manager.motm) OR motorization_manager_is_held(csp_main_motorization_manager.motm) 
THEN
	start_lamp_blink := TRUE;
		start_lamp_on := FALSE;
ELSE
	start_lamp_blink := FALSE;
	start_lamp_on := FALSE;				
END_IF


(* STOP LOGIC *)
IF	machine_is_execute(csp.mch)	
THEN
	stop_lamp_blink := FALSE;
	stop_lamp_on := TRUE;
ELSIF 	motorization_manager_is_stopping(csp_main_motorization_manager.motm)
		OR
		motorization_manager_is_emptying(csp_main_motorization_manager.motm)
THEN
	stop_lamp_blink := TRUE;
	stop_lamp_on := FALSE;
ELSE
	stop_lamp_blink := FALSE;
	stop_lamp_on := FALSE;
END_IF


(* DELAY BEFORE RESET *)

//reset_delay_ton1(IN:=reset_delay_bool , PT:=T#6S , Q=> , ET=> );


IF  csp_case_main_safety_emergency.HMI_Emergency_closed
	AND
	csp_transfer_main_safety_emergency.HMI_Emergency_closed
	OR
	NOT csp_main_accuchange.first_scan_bool
	AND NOT reset_delay_ton_complete1
	THEN
		reset_delay_bool := TRUE; //starts 6 second wait timer
		//reset_delay_ton_complete1 := FALSE;
	ELSE
		reset_delay_bool := FALSE;
END_IF

IF 	reset_delay_ton1.q
THEN
	reset_delay_ton_complete1 := TRUE;
	ELSE
		reset_delay_ton_complete1 := FALSE;
END_IF

reset_delay_ton1(IN:=reset_delay_bool , PT:=T#6S , Q=> , ET=> );

IF reset_delay_bool
	THEN
	timer_restart(6000, reset_tmr);
END_IF


(************************************************************************)

_handle_messages();

_write_output();

powerup := FALSE;

ACTION _handle_messages:
;
END_ACTION

ACTION _handle_process_test:
;
END_ACTION

ACTION _mode_manager:
IF process_mode_req_is_pending(prc)
THEN
    process_apply_mode_req_first_step(prc);
    CASE process_get_mode(prc) OF
        MODE_TO_ABSENT:
			;
        MODE_TO_INACTIVE:
			;
        MODE_TO_TEST:
			;
        MODE_TO_OPERATIONAL:
			powerup := TRUE;
    END_CASE
    process_apply_mode_req_second_step(prc);
END_IF
END_ACTION

ACTION _object_manager:
IF objects_initialization()
THEN
	sub_process_init(
		object_name					:= 'csp_main_services_pushbuttons.prc', 
		process						:= csp_main_services.prc, 
		CONVERSION_this				:= prc);
		
	prc_path 						:= process_get_path(prc);

	
	timer_init(
        object_name                 := CONCAT(prc_path, '_reset_tmr'),
        process                     := prc,
        CONVERSION_this             := reset_tmr);
		
	timer_init(
        object_name                 := CONCAT(prc_path, '_start_tmr'),
        process                     := prc,
        CONVERSION_this             := start_tmr);
		
	digital_check_and_message_init(
		object_name					:= CONCAT(prc_path, '_immediate_stop_dchk'), 
		alarm_if_input_off			:= FALSE, 
		alarm_delay					:= 0, 
		enabled_at_powerup			:= TRUE, 
		individual_reset			:= FALSE, 
		machine_reaction			:= MACHINE_REACTION_EMERGENCY_STOP, 
		typology					:= MESSAGE_TYPOLOGY_ABNORMAL, 
		process						:= prc, 
		CONVERSION_this				:= immediate_stop_dchk);
		
	boolean_init(
		object_name					:= CONCAT(prc_path, '_immediate_stop_bool'), 
		process						:= prc, 
		CONVERSION_this				:= immediate_stop_bool);

	digital_check_add_boolean(
		boolean						:= immediate_stop_bool, 
		CONVERSION_this				:= immediate_stop_dchk);
	
		IF	csp_main_configurator.service_stop_reclassification_present
	THEN
		message_reclassification_init(
			object_name						:= CONCAT(prc_path, '_stop_message_reclassification_instance'),
			process							:= prc,
			CONVERSION_this					:= stop_message_reclassification_instance);

		stop_message_reclassification_instance.get_reclassification_hs := 0;

		filter_init(
			object_name						:= CONCAT(prc_path, '_service_stop_force_unlock_flt'),
			delay_off_on					:= 5000,
			delay_on_off					:= 0,
			process							:= prc,
			CONVERSION_this					:= service_stop_force_unlock_flt);
	END_IF;	
END_IF

IF objects_running()
THEN
	process_cycle(prc);
	digital_check_cycle(immediate_stop_dchk);
	
	IF	csp_main_configurator.service_stop_reclassification_present
	THEN
		message_reclassification_cycle(stop_message_reclassification_instance);

		filter_cycle(
			input			:=	csp_case_main_services_pushbuttons.stop_pressed
								OR
								csp_transfer_main_services_pushbuttons.stop_pressed,
								
			CONVERSION_this := service_stop_force_unlock_flt);
	END_IF
END_IF
END_ACTION

ACTION _read_process_image:
;
END_ACTION

ACTION _read_var_input:
i_reset_button	:= csp_case_main_services_pushbuttons.reset_pressed OR csp_transfer_main_services_pushbuttons.reset_pressed;
i_start_button	:= csp_case_main_services_pushbuttons.start_pressed OR csp_transfer_main_services_pushbuttons.start_pressed;
i_stop_button	:= csp_case_main_services_pushbuttons.stop_pressed OR csp_transfer_main_services_pushbuttons.stop_pressed;
END_ACTION

ACTION _set_runtime_properties:
stop_button_rtrig(CLK:= 
						digital_input_is_active(csp_case_main_services_pushbuttons.stop_di)
						OR
						digital_input_is_active(csp_transfer_main_services_pushbuttons.stop_di)
                  );
				  
stop_dchk_transfer_dvr := digital_check_is_ok(csp_transfer_main_services_pushbuttons.stop_dchk);	

stop_dchk_case_dvr := digital_check_is_ok(csp_case_main_services_pushbuttons.stop_dchk);
					
IF	csp_main_configurator.service_stop_reclassification_present
THEN
	IF	message_reclassification_unlock_guard_enable(stop_message_reclassification_instance)
		OR
		NOT	hmi_is_connected(csp.mch)
		OR
		powerup
		OR
		filter_is_on(service_stop_force_unlock_flt)
	THEN
		unlock_guard_enable_from_reclassification := TRUE;
	END_IF

	IF	machine_is_running(csp.mch)
	THEN
		unlock_guard_enable_from_reclassification := FALSE;
	END_IF
ELSE
	unlock_guard_enable_from_reclassification := TRUE;
END_IF;
END_ACTION

ACTION _write_output:
;
END_ACTION

END_PROGRAM

// ---- Application/CSP/Main/Motorization/csp_main_motorization_manager.TcPOU
(*********************************** G.D S.p.A. - Technical Department ***********************************
============= PROGRAM INFO ============
FOLDER:             TBD
MACHINES INVOLVED:  TBD 

============= DESCRIPTION =============
csp motorization head program

============= REVISIONS ===============
Date		Version	 	Author      	Description             
----------	-------		------------  	--------------------------------------------
2019/04/18 	0000.00	 	M.Grasso		Creation of the PRG

**********************************************************************************************************)
(*$R
	process_ref := prc;
$*)
PROGRAM csp_main_motorization_manager
VAR	
	prc:												process;
	prc_path:											STRING;
	
	motm:												motorization_manager;
	empty_command_motcond:								motorization_conditioner;
	
	suspend_conditions: 								BOOL;
	unsuspend_conditions: 								BOOL;
	suspend_completed: 									BOOL;
	
	reset_production_stats: 							BOOL;
	reset_statistics_cbtn: 								command_button;
	reset_statistics_cbtn_hgos: 						hmi_graphic_object_status;
	debug11: 											BOOL;
	debug10: 											BOOL;
	debug12: 											BOOL;
	Upstream_Wait: 										BOOL;
	Downstream_Wait: 									BOOL;
	reject_command_motcond: 							motorization_conditioner;
	empty_command_velocity: 							LREAL := 10;(*$P $*)
	reject_command_velocity: 							LREAL := 10;(*$P $*)
	debug_Enable_new_conditioners:						BOOL := TRUE;(*$P $*)
END_VAR

VAR CONSTANT
	MACHINE_NOMINAL_VELOCITY_PPM:						INT := 15;
	MACHINE_NOMINAL_VELOCITY_BOUND_PPM:					INT := 20;
	MACHINE_MIN_VELOCITY_PPM:							INT := 5;
	MACHINE_MAX_RELATIVE_OVERSPEED_PPM:					INT := 30;
	MACHINE_ACCELERATION_TIME_S:						LREAL := 5;
	MACHINE_VEL_LIMITED_CHANGE_ACC_DEGPS2:				LREAL := 5; // started at 200
	MACHINE_SERVICE_DECELERATION_TIME_S:				LREAL := 2;
	MACHINE_EMERGENCY_DECELERATION_TIME_S:				LREAL := 0.5;
	MACHINE_ON_PHASE_STOP_SEARCH_SPEED_PPM:				INT := 100;
END_VAR

_read_var_input();

_object_manager();

IF NOT objects_running()
THEN
	RETURN;	
END_IF

_read_process_image();

_mode_manager();

CASE process_get_mode(prc) OF
	MODE_ABSENT,
	MODE_INACTIVE:
		RETURN;
	MODE_TEST:
		_handle_process_test();
END_CASE

_set_runtime_properties();

(********************************* BODY *********************************)
IF csp_case_main_services.dry_cycle_mode
THEN
	motorization_conditioner_deactivate(csp_transfer_infeed_accumulation_level.product_starved_motcond);
END_IF

motorization_conditioner_set_velocity_limit(
	velocity_limit			:= empty_command_velocity,
	CONVERSION_this			:= empty_command_motcond);

IF csp_main_motorization.empty_command
THEN
	motorization_conditioner_velocity_limit_activate(empty_command_motcond);
	motorization_conditioner_deactivate(csp_transfer_infeed_accumulation_level.product_starved_motcond);
ELSE
	motorization_conditioner_velocity_limit_deactivate(empty_command_motcond);
	motorization_conditioner_activate(csp_transfer_infeed_accumulation_level.product_starved_motcond);
END_IF

motorization_conditioner_set_velocity_limit(
	velocity_limit := reject_command_velocity,
	CONVERSION_this := reject_command_motcond);

IF csp_case_transport_virtualMaster.stop_for_reject
THEN
	motorization_conditioner_velocity_limit_activate(reject_command_motcond);
ELSE
	motorization_conditioner_velocity_limit_deactivate(reject_command_motcond);
END_IF

(* Up/Downstream stop Management for OEE Production Counter on Statistics Page *)
suspend_conditions := NOT unsuspend_conditions
							AND csp_main_motorization.execute_bit;

unsuspend_conditions := csp_main_motorization.execute_bit
						AND
						axis_is_moving(csp_case_transport_virtualMaster.axis);
						
IF suspend_conditions
	AND (* Upstream wait conditions *)
	(
		csp_transfer_infeed_accumulation_level.level_status <= CSP_TRANSFER_INFEED_ACCUMULATION_LEVEL_STATUS_MIN
		OR
		csp_case_feed_magazine.hold_request_aml_zone
		OR	
		NOT csp_transfer_upstacker.stack_at_loader
	)	
THEN
	Upstream_Wait := TRUE;
ELSE
	Upstream_Wait := FALSE;
END_IF

IF suspend_conditions
	AND (* Upstream wait conditions *)
	(
		message_is_on(csp_case_discharge_reject_sensors.downstream_backup_di_dchk.alarm_asm.message)
		OR 
		motorization_manager_is_suspended(csp_main_motorization_manager.motm)//message_is_on(csp_main_interface.Cartoner_Stop_Request_aem)	
	)	
THEN
	Downstream_Wait := TRUE;
ELSE
	Downstream_Wait := FALSE;
END_IF				
					


IF suspend_conditions OR debug11(*IN fake Suspend*)
THEN
	machine_set_wait_production_log_lsm_state(TRUE, csp.mch); // This turns the production mode off
	motorization_manager_set_manual_log_state(TRUE, motm); 
	machine_set_production_log_lsm_state(FALSE, csp.mch); //may not be needed but here to be safe
	IF Upstream_Wait OR debug10(* UPSTREAM*)
	THEN
		motorization_manager_set_production_wait_external_up_lsm_state(TRUE,motm);
	ELSIF Downstream_Wait OR debug12(* DOWNSTREAM *) 
	THEN
		motorization_manager_set_production_wait_external_down_lsm_state(TRUE,motm);
	ELSE
		//motorization_manager_set_production_wait_external_operator_lsm_state(TRUE,motm);
	END_IF
ELSE
		motorization_manager_set_manual_log_state(FALSE, motm);
		machine_set_wait_production_log_lsm_state(FALSE, csp.mch);
		machine_set_production_log_lsm_state(TRUE, csp.mch);
END_IF



IF reset_production_stats
THEN
	csp_transfer_infeed_metering_jam.good_carton_count := 0;
	csp_transfer_infeed_metering_jam.waterfall_reject_carton_count := 0;
	csp_transfer_crosspusher.accumulator_reject_carton_count := 0;
	csp_case_transport_virtualMaster.feed_reject_case_count := 0;
	reset_production_stats := FALSE;
END_IF
(************************************************************************)
_handle_messages();

_write_output();

ACTION _handle_messages:
;
END_ACTION

ACTION _handle_process_test:
;
END_ACTION

ACTION _mode_manager:
IF process_mode_req_is_pending(prc)
THEN
    process_apply_mode_req_first_step(prc);
    CASE process_get_mode(prc) OF
        MODE_TO_ABSENT:
			;
        MODE_TO_INACTIVE:
			;
        MODE_TO_TEST:
			;
        MODE_TO_OPERATIONAL:
			;
    END_CASE
    process_apply_mode_req_second_step(prc);
END_IF
END_ACTION

ACTION _object_manager:
IF objects_initialization()
THEN
	sub_process_init(
		object_name								:= 'csp_main_motorization_manager.prc', 
		process									:= csp_main_motorization.prc, 
		CONVERSION_this							:= prc);
		
	prc_path 									:= process_get_path(prc);
	
	motorization_manager_init(
		object_name								:= CONCAT(prc_path, '_motm'), 
		nameplate_nominal_velocity				:= MACHINE_NOMINAL_VELOCITY_PPM, 
		nominal_velocity						:= MACHINE_NOMINAL_VELOCITY_PPM, 
		nominal_velocity_bound					:= MACHINE_NOMINAL_VELOCITY_BOUND_PPM, 
		min_velocity							:= MACHINE_MIN_VELOCITY_PPM, 
		max_relative_overspeed					:= MACHINE_MAX_RELATIVE_OVERSPEED_PPM, 
		units_to_rpm_conversion_factor			:= G_CONV_PPM_TO_DEGPS, 
		acceleration_time						:= MACHINE_ACCELERATION_TIME_S, 
		velocity_limit_change_acceleration		:= MACHINE_VEL_LIMITED_CHANGE_ACC_DEGPS2, 
		service_deceleration_time				:= MACHINE_SERVICE_DECELERATION_TIME_S, 
		emergency_deceleration_time				:= MACHINE_EMERGENCY_DECELERATION_TIME_S, 
		on_phase_stop_type						:= MOTORIZATION_MANAGER_ON_PHASE_STOP_DIRECT, 
		on_phase_stop_search_speed				:= MACHINE_ON_PHASE_STOP_SEARCH_SPEED_PPM, 
		engage_to_main_encoder_when_stopped		:= FALSE, 
		main_motor_axis							:= csp_main_motorization_virtualManager.axis, 
		process									:= prc, 
		CONVERSION_this							:= motm);
		
		
	motorization_conditioner_init(
		object_name								:=	CONCAT(prc_path, '_empty_command_motcond'),
		velocity_limit							:=	empty_command_velocity,
		velocity_limit_active					:=	FALSE,
		idle_handshake_active					:=	FALSE,
		execute_handshake_active				:=	FALSE,
		hold_handshake_active					:=	FALSE,
		suspend_handshake_active				:=	FALSE,
		complete_handshake_active				:=	FALSE,
		abort_handshake_active					:=	FALSE,
		stop_handshake_active					:=	FALSE,
		origin									:=	MOTORIZATION_CONDITIONER_ORIGIN_INTERNAL,
		manager									:=	csp_main_motorization_manager.motm,
		process									:=	prc,
		CONVERSION_this							:=	empty_command_motcond);
		
	motorization_conditioner_init(
		object_name 							:= CONCAT(prc_path, '_reject_command_motcond'),
		velocity_limit 							:= reject_command_velocity,
		velocity_limit_active 					:= FALSE,
		idle_handshake_active 					:= FALSE,
		execute_handshake_active 				:= FALSE,
		hold_handshake_active 					:= FALSE,
		suspend_handshake_active 				:= FALSE,
		complete_handshake_active 				:= FALSE,
		abort_handshake_active 					:= FALSE,
		stop_handshake_active 					:= FALSE,
		origin 									:= MOTORIZATION_CONDITIONER_ORIGIN_INTERNAL,
		manager 								:= csp_main_motorization_manager.motm,
		process									:= prc,
		CONVERSION_this 						:= reject_command_motcond);
END_IF

IF objects_running()
THEN
	process_cycle(prc);
	motorization_manager_cycle(motm);
	motorization_conditioner_cycle(empty_command_motcond);
	motorization_conditioner_cycle(reject_command_motcond);
END_IF
END_ACTION

ACTION _read_process_image:
;
END_ACTION

ACTION _read_var_input:
;
END_ACTION

ACTION _set_runtime_properties:
;
END_ACTION

ACTION _write_output:
;
END_ACTION

END_PROGRAM

// ---- Application/CSP/Case/Main/Services/csp_case_main_services.TcPOU
(********************* G.D S.p.A. - Technical Department *****************************

Date			Version		Author			Description             
----------      -------		-----------		----------------------------------------------
2015/06/30		0000.00		M.Grasso		Initial Release

DESCRIPTION:	

NOTES:        		 

**************************************************************************************)
(*$R process_ref := prc; $*)

PROGRAM csp_case_main_services
VAR
	prc:								process;
	prc_path:							STRING;
	
	reset_output_test:					digital_output;
	
	lights_on_do:						digital_output;
	lights_toggle:						BOOL:=FALSE;(*$P $*)
	dry_cycle_mode:						BOOL:=FALSE; (*$P $*)

	dry_cycle_visu_nvr:            		INT; (*$H_R $*)
	dry_cycle_label_ON_visu_nvr:   		INT; (*$H_R $*)
	dry_cycle_label_OFF_visu_nvr:  		INT; (*$H_R $*)
	
	upstacker_test_visu_nvr:            INT; (*$H_R $*)
	upstacker_test_label_ON_visu_nvr:   INT; (*$H_R $*)
	upstacker_test_label_OFF_visu_nvr:  INT; (*$H_R $*)
	
	cartoner_runout_visu_nvr:           INT; (*$H_R $*)
	end_production_visu_nvr:            INT; (*$H_R $*)
	cartoner_runout_true_cbtn:			command_button;
	cartoner_runout_false_cbtn:			command_button;
	end_production_true_cbtn:			command_button;
	end_production_false_cbtn:			command_button;
	end_production:						BOOL := FALSE;
	empty_cmd_rtrig:					R_TRIG;
	end_production_rtrig:				R_TRIG;
END_VAR

_read_var_input();
_objects_manager();

IF g_application_status <> APPLICATION_STATUS_RUNNING
THEN
	RETURN;
END_IF

_read_process_image();

_mode_manager();

CASE process_get_mode (CONVERSION_this := prc) OF

	MODE_ABSENT,
	MODE_INACTIVE:
		RETURN;

	MODE_TEST:
		_handle_process_test();
END_CASE
_set_runtime_properties();
_visiblity_manager();
(*************************************************************************************
**************************************************************************************)
(*BODY*)

IF descriptor_get_reset_edge(prc.descriptor)
THEN
	digital_output_set(reset_output_test);
ELSE
	digital_output_reset(reset_output_test);
END_IF

IF	csp_main.i_end_job_request
THEN	
	end_production := FALSE;
END_IF

(* LIGHTS ON *)
IF lights_toggle
THEN
	digital_output_set(lights_on_do);
ELSE
	digital_output_reset(lights_on_do);
END_IF

IF command_button_is_pressed(cartoner_runout_true_cbtn)
THEN
	parameter_overwrite_set_bool_value(TRUE,csp_main_motorization.empty_command_overwrite);
END_IF

IF command_button_is_pressed(end_production_true_cbtn)
THEN
	end_production := TRUE;
END_IF

empty_cmd_rtrig(CLK:=csp_main_motorization.empty_command);
end_production_rtrig(CLK:=csp_main_interface.Cartoner_RunOutRequest);

(*************************************************************************************
**************************************************************************************)

_handle_messages();
_write_output();

ACTION _handle_messages:
;
END_ACTION

ACTION _handle_process_test:
;
END_ACTION

ACTION _mode_manager:
IF process_mode_req_is_pending(CONVERSION_this := prc)
THEN
    process_apply_mode_req_first_step(CONVERSION_this := prc);
    CASE process_get_mode(CONVERSION_this := prc) OF
        MODE_TO_ABSENT:
            ;
        MODE_TO_INACTIVE:
            ;
        MODE_TO_TEST:
            ;
        MODE_TO_OPERATIONAL:
            ;
    END_CASE
    process_apply_mode_req_second_step(CONVERSION_this := prc);
END_IF;
END_ACTION

ACTION _objects_manager:
IF objects_initialization()
THEN
    sub_process_init(
	    object_name 	:= 'csp_case_main_services.prc',
        process			:= csp_case_main.prc,
        CONVERSION_this			:= prc);

	prc_path 			:= process_get_path(prc);

	digital_output_init(
		object_name		:= CONCAT(prc_path, '_reset_output_test'),
		polarity_direct	:= TRUE,
		process			:= prc,
		CONVERSION_this			:= reset_output_test);
		
	digital_output_init(
		object_name				:= CONCAT(prc_path, '_lights_on_do'),
		polarity_direct			:= TRUE,
		process					:= prc,
		CONVERSION_this			:= lights_on_do);

	command_button_init(
		object_name				:= CONCAT(prc_path, '_cartoner_runout_true_cbtn'),
		process					:= prc,
		CONVERSION_this			:= cartoner_runout_true_cbtn);
	
	command_button_init(
		object_name				:= CONCAT(prc_path, '_cartoner_runout_false_cbtn'),
		process					:= prc,
		CONVERSION_this			:= cartoner_runout_false_cbtn);
		
	command_button_init(
		object_name				:= CONCAT(prc_path, '_end_production_true_cbtn'),
		process					:= prc,
		CONVERSION_this			:= end_production_true_cbtn);
		
	command_button_init(
		object_name				:= CONCAT(prc_path, '_end_production_false_cbtn'),
		process					:= prc,
		CONVERSION_this			:= end_production_false_cbtn);
		
	end_production_visu_nvr := HMI_OBJECT_STATUS_INVISIBLE;
	command_button_set_status(HMI_OBJECT_STATUS_INVISIBLE,end_production_true_cbtn);
	command_button_set_status(HMI_OBJECT_STATUS_INVISIBLE,end_production_false_cbtn);
	cartoner_runout_visu_nvr := HMI_OBJECT_STATUS_INVISIBLE;
	command_button_set_status(HMI_OBJECT_STATUS_INVISIBLE,cartoner_runout_true_cbtn);
	command_button_set_status(HMI_OBJECT_STATUS_INVISIBLE,cartoner_runout_false_cbtn);

END_IF

IF objects_running()
THEN
	process_cycle(prc);
	command_button_cycle(cartoner_runout_true_cbtn);	
	command_button_cycle(cartoner_runout_false_cbtn);
	command_button_cycle(end_production_true_cbtn);
	command_button_cycle(end_production_false_cbtn);

	
END_IF
END_ACTION

ACTION _read_process_image:
;
END_ACTION

ACTION _read_var_input:
;
END_ACTION

ACTION _set_runtime_properties:
;
END_ACTION

ACTION _visiblity_manager:
IF csp.o_machine_is_stopped
THEN
	dry_cycle_visu_nvr := HMI_OBJECT_STATUS_ON;
	upstacker_test_visu_nvr := HMI_OBJECT_STATUS_ON;
ELSE
	dry_cycle_visu_nvr := HMI_OBJECT_STATUS_INVISIBLE;
	upstacker_test_visu_nvr := HMI_OBJECT_STATUS_INVISIBLE;
END_IF

IF NOT csp.o_machine_is_stopped
THEN
    IF dry_cycle_mode
    THEN
        dry_cycle_label_ON_visu_nvr := HMI_OBJECT_STATUS_ON;
        dry_cycle_label_OFF_visu_nvr := HMI_OBJECT_STATUS_INVISIBLE;
    ELSE
        dry_cycle_label_ON_visu_nvr := HMI_OBJECT_STATUS_INVISIBLE;
        dry_cycle_label_OFF_visu_nvr := HMI_OBJECT_STATUS_ON;
    END_IF
   
    IF csp_transfer_upstacker_sensors.debug_active
    THEN
        upstacker_test_label_ON_visu_nvr := HMI_OBJECT_STATUS_ON;
        upstacker_test_label_OFF_visu_nvr := HMI_OBJECT_STATUS_INVISIBLE;
    ELSE
        upstacker_test_label_ON_visu_nvr := HMI_OBJECT_STATUS_INVISIBLE;
        upstacker_test_label_OFF_visu_nvr := HMI_OBJECT_STATUS_ON;
    END_IF
ELSE
    dry_cycle_label_ON_visu_nvr := HMI_OBJECT_STATUS_INVISIBLE;
    dry_cycle_label_OFF_visu_nvr := HMI_OBJECT_STATUS_INVISIBLE;
    upstacker_test_label_ON_visu_nvr := HMI_OBJECT_STATUS_INVISIBLE;
    upstacker_test_label_OFF_visu_nvr := HMI_OBJECT_STATUS_INVISIBLE;
END_IF

IF end_production_rtrig.Q
THEN
	cartoner_runout_visu_nvr := HMI_OBJECT_STATUS_ON;
	command_button_set_status(HMI_OBJECT_STATUS_ON,cartoner_runout_true_cbtn);
	command_button_set_status(HMI_OBJECT_STATUS_ON,cartoner_runout_false_cbtn);
END_IF

IF empty_cmd_rtrig.Q
THEN
	end_production_visu_nvr := HMI_OBJECT_STATUS_ON;
	command_button_set_status(HMI_OBJECT_STATUS_ON,end_production_true_cbtn);
	command_button_set_status(HMI_OBJECT_STATUS_ON,end_production_false_cbtn);
END_IF

IF command_button_is_pressed(cartoner_runout_true_cbtn) 
	OR command_button_is_pressed(cartoner_runout_false_cbtn)
THEN
		cartoner_runout_visu_nvr := HMI_OBJECT_STATUS_INVISIBLE;
		command_button_set_status(HMI_OBJECT_STATUS_INVISIBLE,cartoner_runout_true_cbtn);
		command_button_set_status(HMI_OBJECT_STATUS_INVISIBLE,cartoner_runout_false_cbtn);
END_IF


IF command_button_is_pressed(end_production_true_cbtn) 
	OR command_button_is_pressed(end_production_false_cbtn)
THEN
		end_production_visu_nvr := HMI_OBJECT_STATUS_INVISIBLE;
		command_button_set_status(HMI_OBJECT_STATUS_INVISIBLE,end_production_true_cbtn);
		command_button_set_status(HMI_OBJECT_STATUS_INVISIBLE,end_production_false_cbtn);
END_IF
END_ACTION

ACTION _write_output:
;
END_ACTION

END_PROGRAM

// ---- Application/CSP/Main/csp_main.TcPOU
(*********************************** G.D S.p.A. - Technical Department ***********************************
============= PROGRAM INFO ============
FOLDER:             TBD
MACHINES INVOLVED:  TBD 

============= DESCRIPTION =============
csp main program

============= REVISIONS ===============
Date		Version	 	Author      	Description             
----------	-------		------------  	--------------------------------------------
2019/04/05 	0000.00	 	M.Grasso		Creation of the PRG

**********************************************************************************************************)
(*$R
	process_ref := prc;
$*)
PROGRAM csp_main
VAR
	prc:												process;
	prc_path:											STRING;
		
	cabinet_ethercat_master:							net_ethercat_master;
	cabinet_transfer_ethercat_master:					net_ethercat_master;
	
	is_SFI:												BOOL := TRUE;
	
END_VAR

VAR_INPUT
	
	i_cabinet_is_running:								BOOL;
	
	i_machine_motor_axis_ref:							POINTER TO axis;
	
	i_csp_data_ref:										POINTER TO csp_customerInterfaces_casePacker;	
	i_start_job_request:								BOOL;	
	i_cycle_enable_request:								BOOL;
	i_end_job_request:									BOOL;	
	i_order_information:								POINTER TO csp_customerInterfaces_order;
	i_product_information:								POINTER TO csp_customerInterfaces_product;
	i_recipe_information:								POINTER TO csp_customerInterfaces_recipe;
	i_current_material_information:						POINTER TO ARRAY[0..14] OF csp_customerInterfaces_material;
	i_next_material_information:						POINTER TO ARRAY[0..14] OF csp_customerInterfaces_material;	
	i_mark_bubd_information:							POINTER TO csp_customerInterfaces_markBUBD;	
	i_cartons_count:									DINT;
	i_next_recipe_information:							POINTER TO csp_customerInterfaces_recipe;
	i_mark_information:									POINTER TO csp_customerInterfaces_mark;	
	i_next_order_information:							POINTER TO csp_customerInterfaces_order;
	i_next_product_information:							POINTER TO csp_customerInterfaces_product;	
	
	(*mch interface*)
	i_cartoner_RunOutComplete:							BOOL;
	i_filler_upstream_coffee:							BOOL;

END_VAR

VAR_OUTPUT
	o_reset_button:										BOOL;
	o_start_button:										BOOL;
END_VAR

_read_var_input();

_object_manager();

IF NOT objects_running()
THEN
	RETURN;	
END_IF

_read_process_image();

_mode_manager();

CASE process_get_mode(prc) of
	MODE_ABSENT,
	MODE_INACTIVE:
		RETURN;
	MODE_TEST:
		_handle_process_test();
END_CASE

_set_runtime_properties();

(********************************* BODY *********************************)

(************************************************************************)

_handle_messages();

_write_output();

ACTION _handle_messages:
;
END_ACTION

ACTION _handle_process_test:
;
END_ACTION

ACTION _mode_manager:
IF process_mode_req_is_pending(prc)
THEN
    process_apply_mode_req_first_step(prc);
    CASE process_get_mode(prc) OF
        MODE_TO_ABSENT:
			;
        MODE_TO_INACTIVE:
			;
        MODE_TO_TEST:
			;
        MODE_TO_OPERATIONAL:
			;
    END_CASE
    process_apply_mode_req_second_step(prc);
END_IF
END_ACTION

ACTION _object_manager:
IF net_initialization()
THEN
		
	net_ethercat_master_init(
		object_name 				:= CONCAT(prc_path, '_cabinet_ethercat_master'), 
		hw_connected				:= TRUE, 
		process						:= prc, 
		CONVERSION_this				:= cabinet_ethercat_master);
		
(*	net_ethercat_master_init(
		object_name 				:= CONCAT(prc_path, '_cabinet_case_ethercat_master'), 
		hw_connected				:= FALSE, 
		process						:= prc, 
		CONVERSION_this				:= cabinet_case_ethercat_master);*)

net_ethercat_master_init(
		object_name 				:= CONCAT(prc_path, '_cabinet_transfer_ethercat_master'), 
		hw_connected				:= TRUE, 
		process						:= prc, 
		CONVERSION_this				:= cabinet_transfer_ethercat_master);				

	
END_IF


IF objects_initialization()
THEN
	process_init(
		object_name					:= 'csp_main.prc', 
		machine						:= csp.mch, 
		CONVERSION_this				:= prc);
		
	prc_path 						:= process_get_path(prc);
	
	hmi_init(
		hmi_is_required				:= TRUE, 
		plc_hmi_protocol_enable		:= FALSE, 
		process						:= prc);
		
	hmi_set_application_version(
		application_name						:= csp_main_configurator.applicaton_name,
		customer								:= csp_main_configurator.customer,
		machine_sequential_number				:= csp_main_configurator.machine_sequential_number,
		application_kickoff_repository_version  := csp_main_configurator.application_kickoff_repository_version,
		safety_version							:= csp_main_configurator.safety_version,
		hardware_version						:= csp_main_configurator.hardware_version,
		software_version						:= csp_main_configurator.software_version);
END_IF

IF objects_running()
THEN
	process_cycle(prc);
END_IF
END_ACTION

ACTION _read_process_image:
;
END_ACTION

ACTION _read_var_input:
i_machine_motor_axis_ref				:= 	ADR(csp_main_motorization_virtualManager.virtual_master_test); //TODO: this will need an update

i_csp_data_ref							:= 	ADR(csp_customerInterfaces.CasePacker);
i_start_job_request						:= 	csp_customerInterfaces.MES.StartJobReq
									   		OR 										//sauro new MES interface
									   		csp_main_phaseManager_startJob.debug_mes_startJobReq;
i_cycle_enable_request					:= 	csp_customerInterfaces.MES.CycleEnable
									  		OR 										//sauro new MES interface
									   		csp_main_phaseManager_startJob.debug_mes_cycleEnable;
i_end_job_request						:= 	csp_customerInterfaces.MES.EndJobReq
	  										OR										//sauro new MES interface
									   		csp_main_phaseManager_end_job.debug_mes_endJobReq;	
i_order_information						:= 	ADR(csp_customerInterfaces.Order);
i_product_information					:= 	ADR(csp_customerInterfaces.Product);
i_recipe_information					:= 	ADR(csp_customerInterfaces.Recipe);
i_current_material_information			:= 	ADR(csp_customerInterfaces.Material);
i_next_material_information				:= 	ADR(csp_customerInterfaces.NextMaterial);	
i_mark_bubd_information					:= 	ADR(csp_customerInterfaces.Mark.BUBD);
i_mark_information						:=  ADR(csp_customerInterfaces.Mark);
i_next_order_information				:=  ADR(csp_customerInterfaces.NextOrder);
i_cartons_count							:=	csp_transfer_infeed_metering_jam.cartons_count;
i_next_recipe_information				:= 	ADR(csp_customerInterfaces.NextRecipe);
i_next_product_information				:= 	ADR(csp_customerInterfaces.NextProduct);
END_ACTION

ACTION _set_runtime_properties:
;
END_ACTION

ACTION _write_output:
o_reset_button	:= csp_case_main_services_pushbuttons.reset_pressed OR csp_transfer_main_services_pushbuttons.reset_pressed;
o_start_button	:= 
	(
		csp_case_main_services_pushbuttons.start_pressed
	 	OR
		csp_transfer_main_services_pushbuttons.start_pressed
	)
	AND
	not csp_main_jogManager.jog_is_active;
END_ACTION

END_PROGRAM

// ---- Application/CSP/Main/csp_main_configurator.TcPOU
(*********************************** G.D S.p.A. - Technical Department ***********************************
============= PROGRAM INFO ============
FOLDER:             TBD
MACHINES INVOLVED:  TBD 

============= DESCRIPTION =============
csp main program

============= REVISIONS ===============
Date		Version	 	Author      	Description             
----------	-------		------------  	--------------------------------------------
2020/05/11 	0000.00	 	M.Grasso		Creation of the PRG

**********************************************************************************************************)
PROGRAM csp_main_configurator
VAR
	prc:												process;
	prc_path:											STRING;
		
	Physical_hw:										BOOL:=TRUE;
	service_stop_reclassification_present: 				BOOL:=TRUE;
	
	applicaton_name:									STRING :='CSP';
	customer:											STRING :='KDP';
	machine_sequential_number:							STRING :='nB4';
	application_kickoff_repository_version:				STRING :='nnnnnnn' ;
	safety_version:										STRING :='000';
	hardware_version:									STRING :='000';
	software_version:									STRING :='000';
	
END_VAR

Physical_hw:=TRUE;
service_stop_reclassification_present:=TRUE;

END_PROGRAM

// ---- Application/CSP/Main/Motorization/csp_main_motorization_virtualManager.TcPOU
(*********************************** G.D S.p.A. - Technical Department ***********************************
============= PROGRAM INFO ============
FOLDER:             TBD
MACHINES INVOLVED:  TBD 

============= DESCRIPTION =============
csp motorization head program

============= REVISIONS ===============
Date		Version	 	Author      	Description             
----------	-------		------------  	--------------------------------------------
2019/04/18 	0000.00	 	M.Grasso		Creation of the PRG

**********************************************************************************************************)
(*$R
	process_ref := prc;
$*)
PROGRAM csp_main_motorization_virtualManager
VAR
	prc:									process;
	prc_path:								STRING;
	
	axis:									axis;
	machine_periodicity_axis:				axis;
	virtual_master_test: 					axis;		
	
	phgen:									phase_generator;				
	

END_VAR

VAR CONSTANT
	MOTOR_MAX_VELOCITY_DEGPS:				LREAL := 9600;
	MOTOR_MAX_ACCELLERATION_DEGPS2:			LREAL := 4800;
	MOTOR_MAX_DECELLERATION_DEGPS2:			LREAL := 4800;
	MOTOR_MAX_JERK_DEGPS3:					LREAL := 100000000; 
	MOTOR_MAX_FOLLOWING_ERROR_DEG:			LREAL := 2;
END_VAR

VAR_OUTPUT
	o_machine_is_moving:					BOOL;
END_VAR

_read_var_input();

_object_manager();

IF NOT objects_running()
THEN
	RETURN;	
END_IF

_read_process_image();

_mode_manager();

CASE process_get_mode(prc) OF
	MODE_ABSENT,
	MODE_INACTIVE:
		RETURN;
	MODE_TEST:
		_handle_process_test();
END_CASE

_set_runtime_properties();

(********************************* BODY *********************************)
(************************************************************************)

_handle_messages();
_feedback();
_write_output();

ACTION _feedback:
;
END_ACTION

ACTION _handle_messages:
;
END_ACTION

ACTION _handle_process_test:
;
END_ACTION

ACTION _mode_manager:
IF process_mode_req_is_pending(prc)
THEN
    process_apply_mode_req_first_step(prc);
    CASE process_get_mode(prc) OF
        MODE_TO_ABSENT:
			;
        MODE_TO_INACTIVE:
			;
        MODE_TO_TEST:
			;
        MODE_TO_OPERATIONAL:
			;
    END_CASE
    process_apply_mode_req_second_step(prc);
END_IF
END_ACTION

ACTION _object_manager:
IF objects_initialization()
THEN
	sub_process_init(
		object_name								:= 'csp_main_motorization_virtualManager.prc', 
		process									:= csp_main_motorization.prc, 
		CONVERSION_this							:= prc);
		
	prc_path 									:= process_get_path(prc);	
	
	(* Motorization virtual axis - 360 degrees -> 1 carton *)	
	axis_init(
		object_name								:= CONCAT(prc_path, '_axis'), 
		axis_type								:= AXIS_TYPE_VIRTUAL, 
		encoder_scaling_factor					:= G_VIRTUAL_ENCODER_SCALING_FACTOR_DEGPINC,
		modulo									:= G_MODULO_360_DEG, 
		process									:= prc, 
		CONVERSION_this							:= axis);
		
	axis_set_max_dynamic(
		reference_velocity						:=	MOTOR_MAX_VELOCITY_DEGPS,
		velocity								:=	MOTOR_MAX_VELOCITY_DEGPS,
		acceleration							:=	MOTOR_MAX_ACCELLERATION_DEGPS2,
		deceleration							:=	MOTOR_MAX_DECELLERATION_DEGPS2,
		jerk									:=	MOTOR_MAX_JERK_DEGPS3,
		following_error							:=	MOTOR_MAX_FOLLOWING_ERROR_DEG,
		CONVERSION_this							:=	axis);
		
	(* Machine periodicity virtual axis - 360 degrees -> number of cartons brand dependent *)	
	axis_init(
		object_name								:= CONCAT(prc_path, '_machine_periodicity_axis'), 
		axis_type								:= AXIS_TYPE_VIRTUAL, 
		encoder_scaling_factor					:= G_VIRTUAL_ENCODER_SCALING_FACTOR_DEGPINC,
		modulo									:= G_MODULO_360_DEG, 
		process									:= prc, 
		CONVERSION_this							:= machine_periodicity_axis);
		
	axis_set_max_dynamic(
		reference_velocity						:= MOTOR_MAX_VELOCITY_DEGPS,
		velocity								:= MOTOR_MAX_VELOCITY_DEGPS,
		acceleration							:= MOTOR_MAX_ACCELLERATION_DEGPS2,
		deceleration							:= MOTOR_MAX_DECELLERATION_DEGPS2,
		jerk									:= MOTOR_MAX_JERK_DEGPS3,
		following_error							:= MOTOR_MAX_FOLLOWING_ERROR_DEG,
		CONVERSION_this							:= machine_periodicity_axis);		
		
	
	//TODO replace with physical servo
	axis_init(
		object_name								:= CONCAT(prc_path, '_virtual_master_test'), 
		axis_type								:= AXIS_TYPE_VIRTUAL, 
		encoder_scaling_factor					:= G_VIRTUAL_ENCODER_SCALING_FACTOR_DEGPINC,
		modulo									:= G_MODULO_360_DEG, 
		process									:= prc, 
		CONVERSION_this							:= virtual_master_test);
		
	axis_set_max_dynamic(
		reference_velocity						:=	MOTOR_MAX_VELOCITY_DEGPS,
		velocity								:=	MOTOR_MAX_VELOCITY_DEGPS,
		acceleration							:=	MOTOR_MAX_ACCELLERATION_DEGPS2,
		deceleration							:=	MOTOR_MAX_DECELLERATION_DEGPS2,
		jerk									:=	MOTOR_MAX_JERK_DEGPS3,
		following_error							:=	MOTOR_MAX_FOLLOWING_ERROR_DEG,
		CONVERSION_this							:=	virtual_master_test);
		
		
	phase_generator_init(
		object_name								:= CONCAT(prc_path, '_phgen'), 
		modulo									:= axis_get_modulo(axis), 
		resolution								:= PHASE_GENERATOR_RESOLUTION_UNIT, 
		axis									:= axis, 
		process									:= prc, 
		CONVERSION_this							:= phgen);	
	
		
END_IF

IF objects_running()
THEN
	process_cycle(prc);
	
	axis_cycle(axis);
	axis_cycle(machine_periodicity_axis);
	axis_cycle(virtual_master_test);
	
	phase_generator_cycle(phgen);
END_IF
END_ACTION

ACTION _read_process_image:
;
END_ACTION

ACTION _read_var_input:
;
END_ACTION

ACTION _set_runtime_properties:
;
END_ACTION

ACTION _write_output:
o_machine_is_moving := axis_is_moving(axis);
END_ACTION

END_PROGRAM

// ---- Application/CSP/Main/Motorization/csp_main_motorization.TcPOU
(*********************************** G.D S.p.A. - Technical Department ***********************************
============= PROGRAM INFO ============
FOLDER:             TBD
MACHINES INVOLVED:  TBD 

============= DESCRIPTION =============
csp motorization head program

============= REVISIONS ===============
Date		Version	 	Author      	Description             
----------	-------		------------  	--------------------------------------------
2019/04/18 	0000.00	 	G.Cera 			Creation of the PRG
2019/04/27	0000.01		G.Cera			Creation of the _connection FSM

**********************************************************************************************************)
(*$R
	process_ref := prc;
$*)
PROGRAM csp_main_motorization
VAR
	prc:												process;
	prc_path:											STRING;
	
	connection_conditions:								BOOL;
	connection_running:									BOOL;
	connection_done:									BOOL;
	connection_timeout:									BOOL;
	connection_status:									csp_main_motorization_connection_status_enum;
	connection_status_mem:								csp_main_motorization_connection_status_enum;
	connection_tmr:										timer;
	connection_done_motcond:							motorization_conditioner;
	
	machine_test_rtrig:									R_TRIG;
	machine_test_ftrig:									F_TRIG;

	fault_aem:											csp_main_motorization_snapshot;	

	motorization_axis_redefined_at_powerup:				BOOL := FALSE;	
	
	empty_command:										BOOL; (*$P $*)
	empty_command_overwrite:							parameter_overwrite;

	STOP_Check: 										BOOL := FALSE;
	
	abort_axes:											BOOL := FALSE; (*$P $*)
	
	execute_BIT: 										BOOL;
	not_execute_BIT: 									BOOL;
	First_Scan: 										BOOL := TRUE;
	abort_axes_auto_reset: 								Ton;
	held_BIT: 											BOOL;
	HOLD_BYPASS: 										BOOL := FALSE;
	unhold_latch_carton_detected: 						BOOL;
	carton_detected_unhold_timer: 						TON;
	counter: 											INT;
	test_cu:											int;
	test_never: 										BOOL;
	abort_axes1: 										BOOL;
END_VAR

VAR CONSTANT
	MULTIGEAR_ACCDEC:									LREAL:= 2000.0;
	CONNECTION_TIMEOUT_S:								INT := 10;
END_VAR

_read_var_input();

_object_manager();

IF 	NOT objects_running()
THEN
	RETURN;	
END_IF

_read_process_image();

_mode_manager();

CASE process_get_mode(prc) OF
	
	MODE_ABSENT,
	MODE_INACTIVE:
		connection_conditions := FALSE;
		connection_done := FALSE;
		connection_status := csp_MAIN_MOTORIZATION_CONNECTION_STATUS_ENUM_CONNECTION_NOT_COMPLETED_STATUS_999;
		RETURN;
		
	MODE_TEST:
		_handle_process_test();
		
END_CASE

_set_runtime_properties();

(********************************* BODY *********************************)

IF First_Scan
	//OR csp_transfer_crosspusher.estop_occured_in_crosspush_reject //this only stays on while the machine is estopped during a reject. Once machine is reset this goes false
THEN
	abort_axes1 := TRUE;
ELSE
	abort_axes1 := FALSE;
END_IF

IF abort_axes
	OR
	abort_axes1
THEN
	test_cu := 1;
	counter := counter +1;
	connection_status := csp_MAIN_MOTORIZATION_CONNECTION_STATUS_ENUM_CONNECTION_NOT_COMPLETED_STATUS_999;
	motorization_axis_redefined_at_powerup := FALSE;
	csp_retain_data.motorization_axis_position := 0;
END_IF


(* TURNS OFF EMPTY COMMAND IF RUN OUT COMPLETE *)
IF process_message_is_on(csp_case_virtualMaster.runout_complete)
	AND machine_is_stopped(csp.mch)
	AND NOT axis_is_moving(csp_main_motorization_virtualManager.axis)
THEN
	parameter_overwrite_set_bool_value(FALSE, empty_command_overwrite);
END_IF

machine_test_ftrig(CLK := machine_is_in_test(csp.mch));
machine_test_rtrig(CLK := machine_is_in_test(csp.mch));

IF	motorization_manager_is_emptying(csp_main_motorization_manager.motm)
THEN
	motorization_manager_empty_done(csp_main_motorization_manager.motm);
END_IF

IF 	machine_test_rtrig.Q
	OR
	machine_test_ftrig.Q
THEN
	connection_conditions := FALSE;
	connection_done := FALSE;
	connection_status := csp_MAIN_MOTORIZATION_CONNECTION_STATUS_ENUM_CONNECTION_NOT_COMPLETED_STATUS_999;
END_IF


IF csp_main_motorization_manager.suspend_conditions
	AND csp_transfer_infeed_accumulation_level_max.di.field.status
THEN
	unhold_latch_carton_detected := TRUE;
END_IF

IF 	csp_transfer_infeed_accumulation_level.level_status >= CSP_TRANSFER_INFEED_ACCUMULATION_LEVEL_STATUS_LOW
	OR carton_detected_unhold_timer.Q
THEN
	unhold_latch_carton_detected := FALSE;
END_IF

carton_detected_unhold_timer(IN:= unhold_latch_carton_detected , PT:=T#20S , Q=>  , ET=> );

	
IF 	csp_case_main_statistics.SHIFT_case_at_loader 
	AND csp_case_main_statistics.SHIFT_case_at_feed
THEN
	motorization_manager_set_velocity_limit_change_acceleration(
		acceleration:= 100,
		conversion_this:= csp_main_motorization_manager.motm);
ELSE
	motorization_manager_set_velocity_limit_change_acceleration(
		acceleration:= 5,
		conversion_this:= csp_main_motorization_manager.motm);
END_IF

IF	(ABS(axis_get_actual_modulo_position(csp_main_motorization_virtualManager.axis) - csp_retain_data.motorization_axis_position) > 1E-2)
 	AND
	motorization_axis_redefined_at_powerup
THEN
	csp_retain_data.motorization_axis_position := axis_get_actual_modulo_position(csp_main_motorization_virtualManager.axis);
END_IF

held_BIT := motorization_manager_is_held(csp_main_motorization_manager.motm);
execute_BIT := motorization_manager_is_execute(csp_main_motorization_manager.motm);
not_execute_BIT := NOT motorization_manager_is_execute(csp_main_motorization_manager.motm);


abort_axes_auto_reset(IN:= abort_axes , PT:=T#2S , Q=>  , ET=> );

IF abort_axes_auto_reset.Q
THEN
	abort_axes := FALSE; //sets abort axes false after 2 seconds of being on to make sure all logic looking at this bit is scanned before truning off
END_IF


connection();
(************************************************************************)

_handle_messages();
_write_output();
First_Scan := FALSE;

ACTION _handle_messages:
IF connection_timeout
THEN
	csp_main_motorization_set_snapshot(
		errorID_1			:= 1, 
		errorID_2			:= 0, 
		errorID_3			:= 0, 
		reason				:= 'CONNECTION TIMEOUT', 
		connection_status	:= connection_status_mem, 
		CONVERSION_this		:= fault_aem);
ELSIF	NOT connection_conditions
		AND
		csp.o_machine_is_running
THEN
	csp_main_motorization_set_snapshot(
		errorID_1			:= 2, 
		errorID_2			:= 0, 
		errorID_3			:= 0, 
		reason				:= 'GROUP NOT READY', 
		connection_status	:= connection_status_mem, 
		CONVERSION_this		:= fault_aem);	
ELSIF	descriptor_get_reset_edge(prc.descriptor)
THEN
	message_reset(fault_aem.message);
END_IF
END_ACTION

ACTION _handle_process_test:
;
END_ACTION

ACTION _mode_manager:
IF process_mode_req_is_pending(prc)
THEN
    process_apply_mode_req_first_step(prc);
    CASE process_get_mode(prc) OF
        MODE_TO_ABSENT:
			;
        MODE_TO_INACTIVE:
			;
        MODE_TO_TEST:
			;
        MODE_TO_OPERATIONAL:
		connection_conditions := FALSE;
		connection_done := FALSE;
		connection_status := csp_MAIN_MOTORIZATION_CONNECTION_STATUS_ENUM_CONNECTION_NOT_COMPLETED_STATUS_999;
    END_CASE
    process_apply_mode_req_second_step(prc);
END_IF
END_ACTION

ACTION _object_manager:
IF objects_initialization()
THEN
	sub_process_init(
		object_name								:= 'csp_main_motorization.prc', 
		process									:= csp_main.prc, 
		CONVERSION_this							:= prc);
			
	prc_path 									:= process_get_path(prc);
	
	(* Connection timer *)
	timer_init(
		object_name								:= CONCAT(prc_path, '_connection_tmr'), 
		process									:= prc, 
		CONVERSION_this							:= connection_tmr);
		
	(* Connection done conditioner *)
	motorization_conditioner_init(
		object_name								:=	CONCAT(prc_path, '_connection_done_motcond'),
		velocity_limit							:=	100.0,
		velocity_limit_active					:=	FALSE,
		idle_handshake_active					:=	FALSE,
		execute_handshake_active				:=	FALSE,
		hold_handshake_active					:=	FALSE,
		suspend_handshake_active				:=	FALSE,
		complete_handshake_active				:=	FALSE,
		abort_handshake_active					:=	FALSE,
		stop_handshake_active					:=	FALSE,
		origin									:=	MOTORIZATION_CONDITIONER_ORIGIN_INTERNAL,
		manager									:=	csp_main_motorization_manager.motm,
		process									:=	prc,
		CONVERSION_this							:=	connection_done_motcond);
		
	(* Snapshot *)
	csp_main_motorization_init_snapshot(
		message_name							:= CONCAT(prc_path, '_fault_aem'), 
		behaviour								:= MESSAGE_BEHAVIOUR_EVENT, 
		reset_timeout							:= 0, 
		disableable								:= FALSE, 
		individual_reset						:= FALSE, 
		machine_reaction						:= MACHINE_REACTION_NO_STOP, 
		typology								:= MESSAGE_TYPOLOGY_GENERIC_1, 
		process									:= prc, 
		CONVERSION_this							:= fault_aem);	
		
		
		
	parameter_overwrite_bool_init(
		object_name								:= CONCAT(prc_path, '_empty_command_overwrite'),
		parameter								:= empty_command,
		process									:= prc,
		CONVERSION_this							:= empty_command_overwrite);
		
END_IF

IF objects_running()
THEN
	process_cycle(prc);
	
	motorization_conditioner_cycle(connection_done_motcond);
END_IF
END_ACTION

ACTION _read_process_image:
;
END_ACTION

ACTION _read_var_input:
;
END_ACTION

ACTION _set_runtime_properties:
;
END_ACTION

ACTION _write_output:
;
END_ACTION

ACTION connection:
connection_conditions :=
	NOT process_message_is_on(fault_aem.message)
	AND
	process_is_ready(prc)
	AND
	process_subtree_is_ready(prc);
	
IF	NOT connection_conditions
	AND
	(
		connection_done
		OR
		connection_running
	)
THEN
	connection_status_mem := connection_status;
	connection_status := csp_MAIN_MOTORIZATION_CONNECTION_STATUS_ENUM_CONNECTION_NOT_COMPLETED_STATUS_999;
END_IF

IF	connection_running
THEN
	IF timer_is_expired(connection_tmr)
	THEN
		connection_status_mem := connection_status;
		connection_timeout := TRUE;
	END_IF
ELSE
	connection_timeout := false;
	timer_restart(CONNECTION_TIMEOUT_S * G_CONV_S_TO_MS, connection_tmr);
END_IF

(* CONNECTION FINITE STATE MACHINE *)
CASE connection_status OF
	
	csp_MAIN_MOTORIZATION_CONNECTION_STATUS_ENUM_IDLE_STATUS_0:
	
		IF	NOT motorization_axis_redefined_at_powerup
			AND
			axis_is_disabled(csp_main_motorization_virtualManager.axis)
			AND
			connection_conditions
		THEN
			connection_running := TRUE;
			connection_status := csp_MAIN_MOTORIZATION_CONNECTION_STATUS_ENUM_VIRTUAL_MANAGER_REDEFINE_POS_REQ_STATUS_20;
		END_IF
	
		
	csp_MAIN_MOTORIZATION_CONNECTION_STATUS_ENUM_AXIS_DISABLE_STATUS_10:
	
		axis_disable(csp_main_motorization_virtualManager.axis);
		
		IF	axis_is_disabled(csp_main_motorization_virtualManager.axis)
		THEN
			connection_status := csp_MAIN_MOTORIZATION_CONNECTION_STATUS_ENUM_VIRTUAL_MANAGER_REDEFINE_POS_REQ_STATUS_20;
		END_IF

		
	csp_MAIN_MOTORIZATION_CONNECTION_STATUS_ENUM_VIRTUAL_MANAGER_REDEFINE_POS_REQ_STATUS_20:
	
		IF	axis_redefine_position(
				position		:= csp_retain_data.motorization_axis_position, 
				mode			:= AXIS_REDEFINE_POSITION_MODE_ABSOLUTE, 
				CONVERSION_this	:= csp_main_motorization_virtualManager.axis)	
		THEN
			connection_status := csp_MAIN_MOTORIZATION_CONNECTION_STATUS_ENUM_VIRTUAL_MANAGER_POS_REDEFINING_STATUS_30;
		END_IF
			
		
	csp_MAIN_MOTORIZATION_CONNECTION_STATUS_ENUM_VIRTUAL_MANAGER_POS_REDEFINING_STATUS_30:
	
		IF 	axis_is_position_redefined(csp_main_motorization_virtualManager.axis)
		THEN
			connection_status := csp_MAIN_MOTORIZATION_CONNECTION_STATUS_ENUM_VIRTUAL_AXIS_ENABLE_STATUS_40;
		ELSIF connection_timeout
		THEN
			connection_running := FALSE;
			connection_status := csp_MAIN_MOTORIZATION_CONNECTION_STATUS_ENUM_AXIS_DISABLE_STATUS_10;
		END_IF	
	
		
	csp_MAIN_MOTORIZATION_CONNECTION_STATUS_ENUM_VIRTUAL_AXIS_ENABLE_STATUS_40:
	
		axis_enable(csp_main_motorization_virtualManager.axis);
		motorization_axis_redefined_at_powerup := TRUE;
		
		IF 	axis_is_standstill(csp_main_motorization_virtualManager.axis)
			AND axis_is_cam_engaged(csp_case_feed_virtualMaster.axis)
			AND axis_is_cam_engaged(csp_case_transport_virtualMaster.axis)
			AND axis_is_cam_engaged(csp_case_loader_virtualMaster.axis)		
			AND axis_is_cam_engaged(csp_case_virtualMaster.axis)		
		THEN	
			connection_status := csp_MAIN_MOTORIZATION_CONNECTION_STATUS_ENUM_CONNECTION_DONE_STATUS_900;
		END_IF
			
					
	csp_MAIN_MOTORIZATION_CONNECTION_STATUS_ENUM_CONNECTION_DONE_STATUS_900:
	
		connection_running := FALSE;
		connection_done := TRUE;
		
		motorization_conditioner_start_done(connection_done_motcond);
	
		
	csp_MAIN_MOTORIZATION_CONNECTION_STATUS_ENUM_CONNECTION_NOT_COMPLETED_STATUS_999:
	
		axis_disable(csp_main_motorization_virtualManager.axis);				
		
		connection_running := FALSE;
		connection_done := FALSE;
		
		IF 	axis_is_disabled(csp_main_motorization_virtualManager.axis)			
		THEN
			connection_status := csp_MAIN_MOTORIZATION_CONNECTION_STATUS_ENUM_IDLE_STATUS_0;
		END_IF
END_CASE
END_ACTION

END_PROGRAM

// ---- Application/CSP/Case/Virtual Master/csp_case_virtualMaster.TcPOU
(*********************************** G.D S.p.A. - Technical Department ***********************************
============= PROGRAM INFO ============
FOLDER:             TBD
MACHINES INVOLVED:  TBD 

============= DESCRIPTION =============
csp machine declaration

============= REVISIONS ===============
Date		Version	 	Author      	Description             
----------	-------		------------  	--------------------------------------------
2019/04/05 	0000.00	 	M.Grasso		Creation of the PRG

**********************************************************************************************************)
(*$R process_ref := prc; $*)
PROGRAM csp_case_virtualMaster
VAR
	
	prc:												process;
	prc_path:											STRING;
	
	fsm_enable_condition:								BOOL := FALSE;
	fsm_next_status:									csp_case_status_enum;
	fsm_status:											csp_case_status_enum;
	
	axis: 												axis;
	phase_position_deg:									LREAL := 0;
	phase_velocity_mmps:								LREAL := 50;
	slave_position_has_been_calculated:					BOOL  := FALSE;
	engage_enable:										BOOL  := TRUE;
	disable_req:										BOOL  := FALSE;
	debug_state_machine:								BOOL  :=FALSE;
	debug_state_machine_one_step:						BOOL  :=FALSE;
	reject_ok:											BOOL  := FALSE;
	reject_busy:										BOOL  := FALSE;
	ready_for_cam:										BOOL  := FALSE;
	cam_engaged:										BOOL  := FALSE;
	phase_enable:										BOOL  := TRUE;
	slave_scaling:										LREAL := 1; 
	master_scaling:										LREAL := 1;
 	load_check_ph_jog:									phase;
	master_offset_phase:								LREAL;
	
	cam_id: 											DINT := LINEAR_CAM;
	axis_calculate_cam_slave_master_position_deg: 		LREAL := 0;
	home_position_master_offset_deg: 					LREAL := 0;
	axis_calculated_cam_slave_position_deg: 			LREAL := 0;
	phase_velocity_degps:								LREAL := 20.0;

	
	Axis_faulted: 										Boolean;
	Axis_faulted_active_dchk: 							digital_check;
	engage_after_estop: 								BOOL := FALSE;
	not_used_11:										BOOL;
	
	
	(* PHASE AND CONNECTION TEST *)
	connection_status: 									csp_case_connection_status_enum;
	connection_status_next: 							csp_case_connection_status_enum;
	connection_done: 									BOOL;
	connection_running: 								BOOL;
	connection_error:									BOOL;
	connection_time_out_tmr:							timer;
	connection_faulted_aem:	 							message;
	connection_conditions:								BOOL;
	connection_done_motcond:							motorization_conditioner;
	connection_motorization_moving:						BOOL;
	
	next_activation_position:							LREAL;	
	activation_position:								LREAL := 0.0;
	
	
	phase_status: 										csp_case_phase_status_enum;
	phase_status_next: 									csp_case_phase_status_enum;
	phase_done: 										BOOL;
	phase_running: 										BOOL;
	phase_error:										BOOL;
	phase_time_out_tmr:									timer;
	phase_faulted_aem:	 								message;
	phase_conditions:									BOOL;
	phase_slave_position:								LREAL;
	
	debug_phase_machine_one_step:						BOOL := FALSE;
	debug_connection_machine_one_step:					BOOL := FALSE;
	debug_immediate_stop_aem:							message;
	debug_immediate_stop:								BOOL;
	
	active_cam:											DINT := DWELL_CAM;
	next_cam:											DINT := DWELL_CAM;
	
	dwell:												BOOL;
	run:												BOOL;
	
	run_test:											BOOL := FALSE;
	
	empty_cycle_count:									INT := 0;
	empty_cycle_runout_input:							INT := 4;
	runout_complete:									message;
	
	run_check_ph: 										phase;
	run_check_ph_deg:									LREAL := 353; (*$P $*)
	
	feed_vm_engaged: 									BOOL;
	transport_vm_engaged: 								BOOL;
	condition1: 										BOOL := FALSE;
	condition2: 										BOOL := FALSE;
	condition3: 										BOOL := False;
	AMR: BOOL;
	engage_count: INT;
END_VAR

VAR CONSTANT
	MOTOR_MAX_VELOCITY_DEGPS:							LREAL := 9600;
	MOTOR_MAX_ACCELLERATION_DEGPS2:						LREAL := 4800;
	MOTOR_MAX_DECELLERATION_DEGPS2:						LREAL := 4800;
	MOTOR_MAX_JERK_DEGPS3:								LREAL := 100000000; 
	MOTOR_MAX_FOLLOWING_ERROR_DEG:						LREAL := 2;
	

END_VAR

_read_var_input();

_object_manager();

IF NOT objects_running()
THEN
	RETURN;	
END_IF

_read_process_image();

_mode_manager();

CASE process_get_mode(prc) OF
	MODE_ABSENT:
		next_cam := DWELL_CAM;
	MODE_INACTIVE:
		RETURN;
	MODE_TEST:
		_handle_process_test();
END_CASE

_set_runtime_properties();

(********************************* BODY *********************************)
(************************************************************************)
IF 	axis_is_moving(csp_main_motorization_virtualManager.axis)
	AND NOT axis_is_ok(FALSE, csp_case_transport_os_trailing.axis)
	AND NOT axis_is_ok(FALSE,csp_case_transport_os_leading.axis)
	AND NOT axis_is_ok(FALSE,csp_case_transport_ls_trailing.axis)
	AND NOT axis_is_ok(FALSE,csp_case_transport_ls_leading.axis)
	AND NOT axis_is_ok(FALSE,csp_case_tr_squaring_ls_leading.axis)
	AND NOT axis_is_ok(FALSE,csp_case_tr_squaring_ls_trailing.axis)
	AND NOT axis_is_ok(FALSE,csp_case_tr_squaring_os_leading.axis)
	AND NOT axis_is_ok(FALSE,csp_case_tr_squaring_os_trailing.axis)
	AND NOT axis_is_ok(FALSE,csp_case_closing_os_horizontal.axis)
	AND NOT axis_is_ok(FALSE,csp_case_closing_os_upper.axis)
	AND NOT axis_is_ok(FALSE,csp_case_closing_os_lower.axis)
	AND NOT axis_is_ok(FALSE,csp_case_closing_ls_horizontal.axis)
	AND NOT axis_is_ok(FALSE,csp_case_closing_ls_upper.axis)
	AND NOT axis_is_ok(FALSE,csp_case_closing_ls_lower.axis)
	AND NOT axis_is_ok(FALSE,csp_case_fc_ls_lower_follower.axis)
	AND NOT axis_is_ok(FALSE,csp_case_fc_ls_lower_spreader.axis)
	AND NOT axis_is_ok(FALSE,csp_case_fc_ls_lower_trailingCloser.axis)
	AND NOT axis_is_ok(FALSE,csp_case_fc_ls_upper_follower.axis)
	AND NOT axis_is_ok(FALSE,csp_case_fc_ls_upper_leadingMinorCloser.axis)
	AND NOT axis_is_ok(FALSE,csp_case_fc_ls_upper_spreader.axis)
	AND NOT axis_is_ok(FALSE,csp_case_fc_os_lower_follower.axis)
	AND NOT axis_is_ok(FALSE,csp_case_fc_os_lower_spreader.axis)
	AND NOT axis_is_ok(FALSE,csp_case_fc_os_upper_follower.axis)
	AND NOT axis_is_ok(FALSE,csp_case_fc_os_upper_spreader.axis)
	AND NOT axis_is_ok(FALSE,csp_case_feed_arm_elbow.axis)
	AND NOT axis_is_ok(FALSE,csp_case_feed_arm_shoulder.axis)
	AND NOT axis_is_ok(FALSE,csp_case_feed_arm_wrist.axis)
	AND NOT axis_is_ok(FALSE,csp_case_feed_shuttle_horizontal.axis)
	AND NOT axis_is_ok(FALSE,csp_case_feed_shuttle_vertical.axis)
	AND NOT axis_is_ok(FALSE,csp_case_loader_guide_downstream.axis)
	//AND not axis_is_ok(FALSE,csp_case_loader_guide_length.axis)
	AND NOT axis_is_ok(FALSE,csp_case_loader_guide_upstream.axis)
	AND NOT axis_is_ok(FALSE,csp_case_loader_pusher.axis)
	//AND not axis_is_ok(FALSE,csp_transfer_infeed_reject_pusher.axis)
	//AND not axis_is_ok(FALSE,csp_transfer_upstacker_downstream.axis)
	//AND not axis_is_ok(FALSE,csp_transfer_upstacker_upstream.axis)
	//AND not axis_is_ok(FALSE,csp_transfer_crosspusher_horizontal.axis)
	//AND not axis_is_ok(FALSE,csp_transfer_crosspusher_vertical.axis)
THEN
    boolean_set(Axis_faulted);
END_IF
  
IF 	machine_is_stop_emergency_active(csp.mch)
	AND motorization_manager_is_stopped(csp_main_motorization_manager.motm)
THEN
	boolean_reset(Axis_faulted);
END_IF

 
 (* USED TO COUNT HOW MANY CYCLES OCCUR BEFORE STOPPING MACHINE *)
IF 	csp_main_motorization.empty_command
	AND csp_transfer_upstacker_sensors.dwell_transfer_empty
	AND phase_edge(csp_case_loader_virtualMaster.load_check_ph)
THEN
	empty_cycle_count := empty_cycle_count + 1;
END_IF

IF 	empty_cycle_count = empty_cycle_runout_input
THEN
	process_message_set(1, 1, 1, runout_complete);
END_IF

IF 	process_message_is_on(runout_complete)
	OR NOT csp_main_motorization.empty_command
THEN
	process_message_reset(runout_complete);
	empty_cycle_count := 0;
END_IF
 
 
(*FSM Control*)
(*disable_req := NOT machine_is_running(csp.mch)
                AND machine_is_stop_emergency_active(csp.mch)
                AND csp_main_motorization_virtualManager.axis.actual_velocity = 0;*)	//_read_var_input
				
IF	machine_is_stop_emergency_active(csp.mch) AND axis_is_cam_engaged(axis) 
THEN
	engage_after_estop := TRUE;
ELSIF NOT machine_is_stop_emergency_active(csp.mch) AND fsm_status = CSP_CASE_STATUS_CAM_ENGAGED 
THEN
	engage_after_estop := FALSE;
END_IF


(* CHECKS TO DETERMINE IF WE CAN INDEX *)
phase_set_data(
	phase				:= run_check_ph_deg,
	delay				:= 0,			
	max_compensation	:= 0,			
	CONVERSION_this		:= run_check_ph);
	
phase_set_data(
	phase				:= csp_case_loader_virtualmaster.load_check_deg,
	delay				:= 0,			
	max_compensation	:= 0,			
	CONVERSION_this		:= load_check_ph_jog);

IF 	axis_is_cam_engaged(csp_case_feed_virtualMaster.axis)
THEN
	feed_vm_engaged :=TRUE;
ELSE
	feed_vm_engaged :=FALSE; 
END_IF
IF 	axis_is_cam_engaged(csp_case_transport_virtualMaster.axis)
THEN
	transport_vm_engaged :=TRUE;
ELSE
	transport_vm_engaged :=FALSE; 
END_IF

(* DECIDES WHETHER TO START OR STOP THE CASE VIRTUAL *)
IF phase_edge(run_check_ph)
THEN
		
	IF 
	( (* USED FOR PRIMING THE CASE SIDE WITH A CASE SO IT IS READY TO LOAD IMMEDIATELY FROM TRANSFER *)
		(
			NOT csp_case_loader.cases_primed 
			AND 
				(
					NOT csp_case_loader.case_at_loader
					OR
					(
						csp_case_loader.case_at_loader
						AND csp_transfer_upstacker.stack_in_case_at_loader
					)
						
				)
		)
		AND NOT csp_case_transport_virtualMaster.stop_for_reject
		AND axis_is_cam_engaged(csp_case_feed_virtualMaster.axis)
		AND NOT message_is_on(csp_case_discharge_reject_sensors.downstream_backup_di_dchk.alarm_asm.message)
		AND NOT message_is_on(csp_main_interface.Cartoner_Stop_Request_aem)
		AND NOT motorization_manager_is_held(csp_main_motorization_manager.motm)//message_is_on(csp_main_interface.Cartoner_Stop_Request_aem)
		//AND NOT csp_case_feed_magazine.suspend_request_aml_zone	
	)
	OR 
	( (* STACK IS READY AND WAITING ON TRANSFER TO RUN (CASE & LOAD AT LOAD SR STEP AND CASE AT FEED SR STEP)*)
		csp_case_loader.case_at_loader
		AND csp_transfer_upstacker.stack_in_case_at_loader
		AND csp_case_loader.cases_primed 
		AND csp_case_fc_ls_upper_leadingMinorCloser.at_upstream_pos
		AND NOT csp_case_transport_virtualMaster.stop_for_reject
		AND axis_is_cam_engaged(csp_case_feed_virtualMaster.axis)
		AND axis_is_cam_engaged(csp_case_transport_virtualMaster.axis)
		AND NOT message_is_on(csp_case_discharge_reject_sensors.downstream_backup_di_dchk.alarm_asm.message)
		AND NOT message_is_on(csp_main_interface.Cartoner_Stop_Request_aem)
		AND NOT motorization_manager_is_held(csp_main_motorization_manager.motm)
		//AND NOT csp_case_feed_magazine.suspend_request_aml_zone	
	)
	OR 
	( (* STACK IS READY AND WAITING ON TRANSFER TO RUN (NO CASE & LOAD AT LOAD SR STEP AND CASE AT FEED SR STEP) *)
		NOT csp_case_loader.case_at_loader
		AND NOT csp_transfer_upstacker.stack_in_case_at_loader
		AND csp_case_loader.cases_primed 
		//AND NOT csp_case_fc_ls_upper_leadingMinorCloser.at_upstream_pos  //removed because no case at loader
		AND NOT csp_case_transport_virtualMaster.stop_for_reject
		AND axis_is_cam_engaged(csp_case_feed_virtualMaster.axis)
		AND axis_is_cam_engaged(csp_case_transport_virtualMaster.axis)
		AND NOT message_is_on(csp_case_discharge_reject_sensors.downstream_backup_di_dchk.alarm_asm.message)
		AND NOT message_is_on(csp_main_interface.Cartoner_Stop_Request_aem)
		AND NOT motorization_manager_is_held(csp_main_motorization_manager.motm)//message_is_on(csp_main_interface.Cartoner_Stop_Request_aem)
		//AND NOT csp_case_feed_magazine.suspend_request_aml_zone	
		)
	OR
	(
		csp_main_motorization.empty_command
		AND csp_transfer_upstacker_sensors.dwell_transfer_empty
		AND empty_cycle_count <= empty_cycle_runout_input
	)
	THEN
		dwell := FALSE;
		run := TRUE;
	ELSE
		run := FALSE;
		dwell := TRUE;
	END_IF
		
END_IF


IF connection_done
THEN 
	motorization_conditioner_start_done(connection_done_motcond);
END_IF

